// TIA Portal V15.1 export
// export: Created 2024-06-21T08:41:19.1954303Z, ExportSetting WithDefaults, DisplayName Totally Integrated Automation Portal, DisplayVersion V15.1 Update 5, DisplayName TIA Portal Openness, DisplayVersion V15.1 Update 5, DisplayName SINAMICS Startdrive Advanced, DisplayVersion V15.1, DisplayName G130, G150, S120, S150, SINAMICS MV, S210, DisplayVersion V15.1, DisplayName G110M, G120, G120C, G120D, G120P, DisplayVersion V15.1, DisplayName STEP 7 Professional, DisplayVersion V15.1 Update 5, DisplayName STEP 7 Safety, DisplayVersion V15.1, DisplayName WinCC Professional, DisplayVersion V15.1 Update 5, DisplayName SIMATIC Visualization Architect, DisplayVersion V15.1
FUNCTION_BLOCK "LGBHoist5Pos-MoviProPN"   // FB6695, FBD
TITLE = LGBMovUnit4Pos-MoviProPN / LGBHoist5Pos-MoviProPN
{ S7_Optimized_Access := 'TRUE' }
AUTHOR : VCC
VERSION : 0.0.0.0
// ============================================================================
// This module is used in applications with a EPOS controlled by a SEW MoviPro frequency converter.
// ============================================================================
// stored: AutoNumber false, IsIECCheckEnabled false, IsRetainMemResEnabled false, MemoryReserve 100, SetENOAutomatically False, UDAEnableTagReadback false
   VAR_INPUT
      I_BeltCheckSensor1 { ExternalAccessible := 'False'; ExternalVisible := 'False'; ExternalWritable := 'False'} : Bool;   // Belt check sensor
      I_BeltCheckSensor2 { ExternalAccessible := 'False'; ExternalVisible := 'False'; ExternalWritable := 'False'} : Bool;   // Belt check sensor
      I_ClutchDetection1 { ExternalAccessible := 'False'; ExternalVisible := 'False'; ExternalWritable := 'False'} : Bool;   // Clutch detection
      I_ClutchDetection2 { ExternalAccessible := 'False'; ExternalVisible := 'False'; ExternalWritable := 'False'} : Bool;   // Clutch detection
      I_Position1Begin { ExternalAccessible := 'False'; ExternalVisible := 'False'; ExternalWritable := 'False'} : Bool;   // Start Move To Position
      I_Position2Begin { ExternalAccessible := 'False'; ExternalVisible := 'False'; ExternalWritable := 'False'} : Bool;   // Start Move To Position
      I_Position3Begin { ExternalAccessible := 'False'; ExternalVisible := 'False'; ExternalWritable := 'False'} : Bool;   // Start Move To Position
      I_Position4Begin { ExternalAccessible := 'False'; ExternalVisible := 'False'; ExternalWritable := 'False'} : Bool;   // Start Move To Position
      I_Position5Begin { ExternalAccessible := 'False'; ExternalVisible := 'False'; ExternalWritable := 'False'} : Bool;   // Start Move To Position
      I_PositionMaintenanceBegin { ExternalAccessible := 'False'; ExternalVisible := 'False'; ExternalWritable := 'False'} : Bool;   // Start Move To Position / Start Move To Position Maintenance
      I_InterlockPos1 { ExternalAccessible := 'False'; ExternalVisible := 'False'; ExternalWritable := 'False'} : Bool;   // Interlock Pos1
      I_InterlockPos2 { ExternalAccessible := 'False'; ExternalVisible := 'False'; ExternalWritable := 'False'} : Bool;   // Interlock Pos2
      I_InterlockPos3 { ExternalAccessible := 'False'; ExternalVisible := 'False'; ExternalWritable := 'False'} : Bool;   // Interlock Pos3
      I_InterlockPos4 { ExternalAccessible := 'False'; ExternalVisible := 'False'; ExternalWritable := 'False'} : Bool;   // Interlock Pos4
      I_InterlockPos5 { ExternalAccessible := 'False'; ExternalVisible := 'False'; ExternalWritable := 'False'} : Bool;   // Interlock Pos4 / Interlock Pos5
      I_InterlockPosMaintenance { ExternalAccessible := 'False'; ExternalVisible := 'False'; ExternalWritable := 'False'} : Bool;   // Interlock Pos4 / Interlock Pos Maintenance
      I_InterlockJog { ExternalAccessible := 'False'; ExternalVisible := 'False'; ExternalWritable := 'False'} : Bool;   // Interlock Jog -/+ / Interlock jog set
      I_InterlockReferencing { ExternalAccessible := 'False'; ExternalVisible := 'False'; ExternalWritable := 'False'} : Bool;   // Interlock Referencing / Interlock jog set
      I_LocalPBSet { ExternalAccessible := 'False'; ExternalVisible := 'False'; ExternalWritable := 'False'} : Bool;   // Push button for manual movememt (on local panel)
      I_LocalPBRes { ExternalAccessible := 'False'; ExternalVisible := 'False'; ExternalWritable := 'False'} : Bool;   // Push button for manual movememt Reset(on local panel)
      I_MotorProtection { ExternalAccessible := 'False'; ExternalVisible := 'False'; ExternalWritable := 'False'} : Bool;   // Motor protection
      I_ReleaseBrake { ExternalAccessible := 'False'; ExternalVisible := 'False'; ExternalWritable := 'False'} : Bool;   // Release brake
      I_Distance { ExternalAccessible := 'False'; ExternalVisible := 'False'; ExternalWritable := 'False'} : DInt;   // Current distance / Current distance in the current resolution under consideration of offset. Depending on resolution, one digit corresponds to 0.1 to 100 mm.
      I_SafetyOk { ExternalAccessible := 'False'; ExternalVisible := 'False'; ExternalWritable := 'False'} : Bool;   // Safety Ok
      I_MotionStopOk { ExternalAccessible := 'False'; ExternalVisible := 'False'; ExternalWritable := 'False'} : Bool;   // Safety Ok / The motion stop is Ok
      I_AutoSpeed { ExternalAccessible := 'False'; ExternalVisible := 'False'; ExternalWritable := 'False'} : Int;   // Auto speed Value
      I_ManualSpeed { ExternalAccessible := 'False'; ExternalVisible := 'False'; ExternalWritable := 'False'} : Int;   // Manual speed Value
      I_SafetyStatus { ExternalAccessible := 'False'; ExternalVisible := 'False'; ExternalWritable := 'False'} : Word;   // Safety Status
      I_SafetyControl { ExternalAccessible := 'False'; ExternalVisible := 'False'; ExternalWritable := 'False'} : Word;   // Safety Control Word
   END_VAR
   VAR_OUTPUT
      O_Active { ExternalAccessible := 'False'; ExternalVisible := 'False'; ExternalWritable := 'False'} : Bool;   // Machine is active
      O_Position1Finished { ExternalAccessible := 'False'; ExternalVisible := 'False'; ExternalWritable := 'False'} : Bool;   // Position 1 finished
      O_Position2Finished { ExternalAccessible := 'False'; ExternalVisible := 'False'; ExternalWritable := 'False'} : Bool;   // Position 2 finished
      O_Position3Finished { ExternalAccessible := 'False'; ExternalVisible := 'False'; ExternalWritable := 'False'} : Bool;   // Position 3 finished
      O_Position4Finished { ExternalAccessible := 'False'; ExternalVisible := 'False'; ExternalWritable := 'False'} : Bool;   // Position 4 finished
      O_Position5Finished { ExternalAccessible := 'False'; ExternalVisible := 'False'; ExternalWritable := 'False'} : Bool;   // Position 4 finished / Position 5 finished
      O_PositionMaintenanceFinished { ExternalAccessible := 'False'; ExternalVisible := 'False'; ExternalWritable := 'False'} : Bool;   // Position 4 finished / Position Maintenance finished
      O_InPosition1 { ExternalAccessible := 'False'; ExternalVisible := 'False'; ExternalWritable := 'False'} : Bool;   // In Position 1
      O_InPosition2 { ExternalAccessible := 'False'; ExternalVisible := 'False'; ExternalWritable := 'False'} : Bool;   // In Position 2
      O_InPosition3 { ExternalAccessible := 'False'; ExternalVisible := 'False'; ExternalWritable := 'False'} : Bool;   // In Position 3
      O_InPosition4 { ExternalAccessible := 'False'; ExternalVisible := 'False'; ExternalWritable := 'False'} : Bool;   // In Position 4
      O_InPosition5 { ExternalAccessible := 'False'; ExternalVisible := 'False'; ExternalWritable := 'False'} : Bool;   // In Position 4 / In Position 5
      O_InPositionMaintenance { ExternalAccessible := 'False'; ExternalVisible := 'False'; ExternalWritable := 'False'} : Bool;   // In Position 4 / In Position Maintenance
      O_ActualPosition { ExternalAccessible := 'False'; ExternalVisible := 'False'; ExternalWritable := 'False'} : DInt;   // Actual position
      O_LEDPosition1 { ExternalAccessible := 'False'; ExternalVisible := 'False'; ExternalWritable := 'False'} : Bool;   // Ledindication / Led indication for Position1
      O_LEDPosition2 { ExternalAccessible := 'False'; ExternalVisible := 'False'; ExternalWritable := 'False'} : Bool;   // Ledindication / Led indication for Position2
      O_LEDPosition3 { ExternalAccessible := 'False'; ExternalVisible := 'False'; ExternalWritable := 'False'} : Bool;   // Ledindication / Led indication for Position3
      O_LEDPosition4 { ExternalAccessible := 'False'; ExternalVisible := 'False'; ExternalWritable := 'False'} : Bool;   // Ledindication / Led indication for Position4
      O_LEDPosition5 { ExternalAccessible := 'False'; ExternalVisible := 'False'; ExternalWritable := 'False'} : Bool;   // Ledindication / Led indication for Position5
      O_AlarmABCondition { ExternalAccessible := 'False'; ExternalVisible := 'False'; ExternalWritable := 'False'} : Bool;   // Alarm AB condition
      O_AlarmA { ExternalAccessible := 'False'; ExternalVisible := 'False'; ExternalWritable := 'False'} : Bool;   // Summation Alarm A
      O_AlarmB { ExternalAccessible := 'False'; ExternalVisible := 'False'; ExternalWritable := 'False'} : Bool;   // Summation Alarm B
      O_AlarmC { ExternalAccessible := 'False'; ExternalVisible := 'False'; ExternalWritable := 'False'} : Bool;   // Summation Alarm C
      O_AlarmD { ExternalAccessible := 'False'; ExternalVisible := 'False'; ExternalWritable := 'False'} : Bool;   // Summation Alarm D
      H_AlarmDWord { ExternalAccessible := 'False'; ExternalVisible := 'False'; ExternalWritable := 'False'} : DWord;   // HMI Animation of the alarms
      H_AlarmDWord2 { ExternalAccessible := 'False'; ExternalVisible := 'False'; ExternalWritable := 'False'} : DWord;   // HMI Animation of the alarms
   END_VAR
   VAR_IN_OUT
      IO_Modes : "Modes";   // Modes
      H_HMI : "H_HMI";   // Animation
      "H_GBHoist5Pos-MoviProPN" : "H_GBHoist5Pos-MoviProPN";   // Animation
      C_Config : "Hoist5Pos-MoviProPNConfig";   // Config
   END_VAR
   VAR
      AA_MotorProtection { ExternalAccessible := 'False'; ExternalVisible := 'False'; ExternalWritable := 'False'} : Bool;   // Motorprotection Tripped / Motorprotection Not Ok
      AA_SafetySwitch { ExternalAccessible := 'False'; ExternalVisible := 'False'; ExternalWritable := 'False'} : Bool;   // Safety Switch Not Ok
      AB_STO { ExternalAccessible := 'False'; ExternalVisible := 'False'; ExternalWritable := 'False'} : Bool;   // Safety Switch Not Ok / Safety output to drive is active but no response from drive that the safety is ok
      AB_DriveNoResponse { ExternalAccessible := 'False'; ExternalVisible := 'False'; ExternalWritable := 'False'} : Bool;   // Alarm Frequency Control / Alarm Frequency Control - No Responce from Drive (live bit)
      AB_DriveAlarm { ExternalAccessible := 'False'; ExternalVisible := 'False'; ExternalWritable := 'False'} : Bool;   // Frequency Control / Alarm Frequency Control
      AD_DriveWarning { ExternalAccessible := 'False'; ExternalVisible := 'False'; ExternalWritable := 'False'} : Bool;   // Warning Frequency Control / Warning
      AA_BeltCheck1 { ExternalAccessible := 'False'; ExternalVisible := 'False'; ExternalWritable := 'False'} : Bool;   // Remkontroll 1 / Belt Control Detection 1
      AA_BeltCheck2 { ExternalAccessible := 'False'; ExternalVisible := 'False'; ExternalWritable := 'False'} : Bool;   // Remkontroll 2 / Belt Control Detection 2
      AB_ClutchDetection { ExternalAccessible := 'False'; ExternalVisible := 'False'; ExternalWritable := 'False'} : Bool;   // Remkontroll 2 / No or both clutches engaged
      AB_OverTravelSet { ExternalAccessible := 'False'; ExternalVisible := 'False'; ExternalWritable := 'False'} : Bool;   // Overtravel Set
      AB_OverTravelRes { ExternalAccessible := 'False'; ExternalVisible := 'False'; ExternalWritable := 'False'} : Bool;   // Overtravel Reset
      AB_EncDifference { ExternalAccessible := 'False'; ExternalVisible := 'False'; ExternalWritable := 'False'} : Bool;   // Profinet <-> SSI encoder difference alarm
      AC_OvtPos1 { ExternalAccessible := 'False'; ExternalVisible := 'False'; ExternalWritable := 'False'} : Bool;   // Timeout Pos 1 / TimeOut to Position 1
      AC_OvtPos2 { ExternalAccessible := 'False'; ExternalVisible := 'False'; ExternalWritable := 'False'} : Bool;   // Timeout Pos 2 / TimeOut to Position 2
      AC_OvtPos3 { ExternalAccessible := 'False'; ExternalVisible := 'False'; ExternalWritable := 'False'} : Bool;   // Timeout Pos 3 / TimeOut to Position 3
      AC_OvtPos4 { ExternalAccessible := 'False'; ExternalVisible := 'False'; ExternalWritable := 'False'} : Bool;   // Timeout Pos 4 / TimeOut to Position 4
      AC_OvtPos5 { ExternalAccessible := 'False'; ExternalVisible := 'False'; ExternalWritable := 'False'} : Bool;   // Timeout Pos 4 / TimeOut to Position 5
      AC_OvtPosMaintenance { ExternalAccessible := 'False'; ExternalVisible := 'False'; ExternalWritable := 'False'} : Bool;   // Timeout Pos 4 / TimeOut to Position Maintenance
      AC_KeepPos1 { ExternalAccessible := 'False'; ExternalVisible := 'False'; ExternalWritable := 'False'} : Bool;   // Position Supervision / Lost Position 1
      AC_KeepPos2 { ExternalAccessible := 'False'; ExternalVisible := 'False'; ExternalWritable := 'False'} : Bool;   // Position Supervision / Lost Position 2
      AC_KeepPos3 { ExternalAccessible := 'False'; ExternalVisible := 'False'; ExternalWritable := 'False'} : Bool;   // Position Supervision / Lost Position 3
      AC_KeepPos4 { ExternalAccessible := 'False'; ExternalVisible := 'False'; ExternalWritable := 'False'} : Bool;   // Position Supervision / Lost Position 4
      AC_KeepPos5 { ExternalAccessible := 'False'; ExternalVisible := 'False'; ExternalWritable := 'False'} : Bool;   // Position Supervision / Lost Position 5
      AD_IntlkPos1 { ExternalAccessible := 'False'; ExternalVisible := 'False'; ExternalWritable := 'False'} : Bool;   // Interlock Not Ok / Interlock Position 1
      AD_IntlkPos2 { ExternalAccessible := 'False'; ExternalVisible := 'False'; ExternalWritable := 'False'} : Bool;   // Interlock Not Ok / Interlock Position 2
      AD_IntlkPos3 { ExternalAccessible := 'False'; ExternalVisible := 'False'; ExternalWritable := 'False'} : Bool;   // Interlock Not Ok / Interlock Position 3
      AD_IntlkPos4 { ExternalAccessible := 'False'; ExternalVisible := 'False'; ExternalWritable := 'False'} : Bool;   // Interlock Not Ok / Interlock Position 4
      AD_IntlkPos5 { ExternalAccessible := 'False'; ExternalVisible := 'False'; ExternalWritable := 'False'} : Bool;   // Interlock Not Ok / Interlock Position 5
      AD_IntlkPosMaintenance { ExternalAccessible := 'False'; ExternalVisible := 'False'; ExternalWritable := 'False'} : Bool;   // Interlock Not Ok / Interlock Position Maintenance
      AD_IntrlJogMode { ExternalAccessible := 'False'; ExternalVisible := 'False'; ExternalWritable := 'False'} : Bool;   // Interlock Jog Mode / Interlock Not Ok for jog set
      AD_IntrlReferencing { ExternalAccessible := 'False'; ExternalVisible := 'False'; ExternalWritable := 'False'} : Bool;   // Interlock Referencing / Interlock Not Ok for jog set
      AD_JogModeActive { ExternalAccessible := 'False'; ExternalVisible := 'False'; ExternalWritable := 'False'} : Bool;   // Jog Mode is active
      AD_ReferencingActive { ExternalAccessible := 'False'; ExternalVisible := 'False'; ExternalWritable := 'False'} : Bool;   // Referencing is active
      AD_EmergencyModeActive { ExternalAccessible := 'False'; ExternalVisible := 'False'; ExternalWritable := 'False'} : Bool;   // Emergency Mode is active
      AD_MotionStop { ExternalAccessible := 'False'; ExternalVisible := 'False'; ExternalWritable := 'False'} : Bool;   // Motion Stop
      SafetyOk { ExternalAccessible := 'False'; ExternalVisible := 'False'; ExternalWritable := 'False'} : Bool;   // Safety Ok
      AlarmA { ExternalAccessible := 'False'; ExternalVisible := 'False'; ExternalWritable := 'False'} : Bool;   // Alarm A
      AlarmB { ExternalAccessible := 'False'; ExternalVisible := 'False'; ExternalWritable := 'False'} : Bool;   // Alarm B
      AlarmC { ExternalAccessible := 'False'; ExternalVisible := 'False'; ExternalWritable := 'False'} : Bool;   // Alarm C
      AlarmD { ExternalAccessible := 'False'; ExternalVisible := 'False'; ExternalWritable := 'False'} : Bool;   // Alarm D
      AlarmABCondition { ExternalAccessible := 'False'; ExternalVisible := 'False'; ExternalWritable := 'False'} : Bool;   // Alarm AB Condition
      Referencing { ExternalAccessible := 'False'; ExternalVisible := 'False'; ExternalWritable := 'False'} : Bool;   // Activate Calibration
      EmergencyMode { ExternalAccessible := 'False'; ExternalVisible := 'False'; ExternalWritable := 'False'} : Bool;   // Emergency mode (without encoder)
      DriveMode { ExternalAccessible := 'False'; ExternalVisible := 'False'; ExternalWritable := 'False'} : Bool;   // 1 = direct setpoint / 0 = Jogmode
      JogMode { ExternalAccessible := 'False'; ExternalVisible := 'False'; ExternalWritable := 'False'} : Bool;   // 1= jog mode / 0= normal mode
      EPosCmdPos1 { ExternalAccessible := 'False'; ExternalVisible := 'False'; ExternalWritable := 'False'} : Bool;   // Cmd Pos 1 Direction
      EPosCmdPos2 { ExternalAccessible := 'False'; ExternalVisible := 'False'; ExternalWritable := 'False'} : Bool;   // Cmd Pos 2 Direction
      EPosCmdPos3 { ExternalAccessible := 'False'; ExternalVisible := 'False'; ExternalWritable := 'False'} : Bool;   // Cmd Pos 3 Direction
      EPosCmdPos4 { ExternalAccessible := 'False'; ExternalVisible := 'False'; ExternalWritable := 'False'} : Bool;   // Cmd Pos 4 Direction
      EPosCmdPos5 { ExternalAccessible := 'False'; ExternalVisible := 'False'; ExternalWritable := 'False'} : Bool;   // Cmd Pos 5 Direction / Cmd Pos 4 Direction
      EPosCmdPosMaintenance { ExternalAccessible := 'False'; ExternalVisible := 'False'; ExternalWritable := 'False'} : Bool;   // Cmd Pos Maintenance Direction / Cmd Pos 4 Direction
      MotorLoopActive { ExternalAccessible := 'False'; ExternalVisible := 'False'; ExternalWritable := 'False'} : Bool;   // Motor Loop Active
      BeltCheck1AlmCond { ExternalAccessible := 'False'; ExternalVisible := 'False'; ExternalWritable := 'False'} : Bool;   // Belt check alarm condition
      BeltCheck2AlmCond { ExternalAccessible := 'False'; ExternalVisible := 'False'; ExternalWritable := 'False'} : Bool;   // Belt check alarm condition
      ClutchDetectionAlmCond { ExternalAccessible := 'False'; ExternalVisible := 'False'; ExternalWritable := 'False'} : Bool;   // Belt check alarm condition
      OverTravelSetAlmCond { ExternalAccessible := 'False'; ExternalVisible := 'False'; ExternalWritable := 'False'} : Bool;   // Overtravel set alarm condition
      OverTravelResAlmCond { ExternalAccessible := 'False'; ExternalVisible := 'False'; ExternalWritable := 'False'} : Bool;   // Overtravel reset alarm condition
      MotorLoopAlarmCond { ExternalAccessible := 'False'; ExternalVisible := 'False'; ExternalWritable := 'False'} : Bool;   // Motor loop alarm condition
      EncDifferenceAlmCond { ExternalAccessible := 'False'; ExternalVisible := 'False'; ExternalWritable := 'False'} : Bool;   // Belt check alarm condition / Encoder Diff alarm condition
      ManReqIndexPos1 { ExternalAccessible := 'False'; ExternalVisible := 'False'; ExternalWritable := 'False'} : Bool;   // Manual request position 1
      ManReqIndexPos2 { ExternalAccessible := 'False'; ExternalVisible := 'False'; ExternalWritable := 'False'} : Bool;   // Manual request position 2
      ManReqIndexPos3 { ExternalAccessible := 'False'; ExternalVisible := 'False'; ExternalWritable := 'False'} : Bool;   // Manual request position 3
      ManReqIndexPos4 { ExternalAccessible := 'False'; ExternalVisible := 'False'; ExternalWritable := 'False'} : Bool;   // Manual request position 4
      ManReqIndexPos5 { ExternalAccessible := 'False'; ExternalVisible := 'False'; ExternalWritable := 'False'} : Bool;   // Manual request position 5 / Manual request position 4
      ManReqIndexPosMaintenance { ExternalAccessible := 'False'; ExternalVisible := 'False'; ExternalWritable := 'False'} : Bool;   // Manual request position Maintenance / Manual request position 4
      CmdPos1 { ExternalAccessible := 'False'; ExternalVisible := 'False'; ExternalWritable := 'False'} : Bool;   // Index position 1 command
      CmdPos2 { ExternalAccessible := 'False'; ExternalVisible := 'False'; ExternalWritable := 'False'} : Bool;   // Index position 2 command
      CmdPos3 { ExternalAccessible := 'False'; ExternalVisible := 'False'; ExternalWritable := 'False'} : Bool;   // Index position 3 command
      CmdPos4 { ExternalAccessible := 'False'; ExternalVisible := 'False'; ExternalWritable := 'False'} : Bool;   // Index position 4 command
      CmdPos5 { ExternalAccessible := 'False'; ExternalVisible := 'False'; ExternalWritable := 'False'} : Bool;   // Index position 4 command / Index position 5 command
      CmdPosMaintenance { ExternalAccessible := 'False'; ExternalVisible := 'False'; ExternalWritable := 'False'} : Bool;   // Index position 4 command / Index position Maintenance command
   END_VAR
   VAR RETAIN
      InPos1 { ExternalAccessible := 'False'; ExternalVisible := 'False'; ExternalWritable := 'False'} : Bool;   // In position 1
      InPos2 { ExternalAccessible := 'False'; ExternalVisible := 'False'; ExternalWritable := 'False'} : Bool;   // In position 2
      InPos3 { ExternalAccessible := 'False'; ExternalVisible := 'False'; ExternalWritable := 'False'} : Bool;   // In position 3
      InPos4 { ExternalAccessible := 'False'; ExternalVisible := 'False'; ExternalWritable := 'False'} : Bool;   // In position 4
      InPos5 { ExternalAccessible := 'False'; ExternalVisible := 'False'; ExternalWritable := 'False'} : Bool;   // In position 4 / In position 5
      InPosMaintenance { ExternalAccessible := 'False'; ExternalVisible := 'False'; ExternalWritable := 'False'} : Bool;   // In position 4 / In position Maintenance
   END_VAR
   VAR
      InterlockPos1 { ExternalAccessible := 'False'; ExternalVisible := 'False'; ExternalWritable := 'False'} : Bool;   // Interlock Pos1
      InterlockPos2 { ExternalAccessible := 'False'; ExternalVisible := 'False'; ExternalWritable := 'False'} : Bool;   // Interlock Pos2
      InterlockPos3 { ExternalAccessible := 'False'; ExternalVisible := 'False'; ExternalWritable := 'False'} : Bool;   // Interlock Pos3
      InterlockPos4 { ExternalAccessible := 'False'; ExternalVisible := 'False'; ExternalWritable := 'False'} : Bool;   // Interlock Pos4
      InterlockPos5 { ExternalAccessible := 'False'; ExternalVisible := 'False'; ExternalWritable := 'False'} : Bool;   // Interlock Pos4 / Interlock Pos5
      InterlockPosMaintenance { ExternalAccessible := 'False'; ExternalVisible := 'False'; ExternalWritable := 'False'} : Bool;   // Interlock Pos4 / Interlock PosMaintenance
      InterlockJog { ExternalAccessible := 'False'; ExternalVisible := 'False'; ExternalWritable := 'False'} : Bool;   // Interlock Jog -/+ / Interlock jog set
      InterlockReferencing { ExternalAccessible := 'False'; ExternalVisible := 'False'; ExternalWritable := 'False'} : Bool;   // Interlock Referencing / Interlock jog set
      ReadyForOperation { ExternalAccessible := 'False'; ExternalVisible := 'False'; ExternalWritable := 'False'} : Bool;   // Ready for operation
      EPOSInPosition { ExternalAccessible := 'False'; ExternalVisible := 'False'; ExternalWritable := 'False'} : Bool;   // Target Position reached
      AxisHomed { ExternalAccessible := 'False'; ExternalVisible := 'False'; ExternalWritable := 'False'} : Bool;   // Axis homed
      AxisMoving { ExternalAccessible := 'False'; ExternalVisible := 'False'; ExternalWritable := 'False'} : Bool;   // Axis moving in any direction
      InStandstill { ExternalAccessible := 'False'; ExternalVisible := 'False'; ExternalWritable := 'False'} : Bool;   // Axis in standstill
      Jog { ExternalAccessible := 'False'; ExternalVisible := 'False'; ExternalWritable := 'False'} : Bool;   // Activate Jog Mode
      Start { ExternalAccessible := 'False'; ExternalVisible := 'False'; ExternalWritable := 'False'} : Bool;   // Start command to motor
      SetpointSpeed { ExternalAccessible := 'False'; ExternalVisible := 'False'; ExternalWritable := 'False'} : Int;   // Setpoint speed
      LastCmd1 { ExternalAccessible := 'False'; ExternalVisible := 'False'; ExternalWritable := 'False'} : Bool;   // Last Command to Drive Is Pos 1
      LastCmd2 { ExternalAccessible := 'False'; ExternalVisible := 'False'; ExternalWritable := 'False'} : Bool;   // Last Command to Drive Is Pos 2
      LastCmd3 { ExternalAccessible := 'False'; ExternalVisible := 'False'; ExternalWritable := 'False'} : Bool;   // Last Command to Drive Is Pos 3
      LastCmd4 { ExternalAccessible := 'False'; ExternalVisible := 'False'; ExternalWritable := 'False'} : Bool;   // Last Command to Drive Is Pos 4
      LastCmd5 { ExternalAccessible := 'False'; ExternalVisible := 'False'; ExternalWritable := 'False'} : Bool;   // Last Command to Drive Is Pos 4 / Last Command to Drive Is Pos 5
      AlmCondKeepPos1 { ExternalAccessible := 'False'; ExternalVisible := 'False'; ExternalWritable := 'False'} : Bool;   // Alarm Condition Keep Position 1
      AlmCondKeepPos2 { ExternalAccessible := 'False'; ExternalVisible := 'False'; ExternalWritable := 'False'} : Bool;   // Alarm Condition Keep Position 2
      AlmCondKeepPos3 { ExternalAccessible := 'False'; ExternalVisible := 'False'; ExternalWritable := 'False'} : Bool;   // Alarm Condition Keep Position 3
      AlmCondKeepPos4 { ExternalAccessible := 'False'; ExternalVisible := 'False'; ExternalWritable := 'False'} : Bool;   // Alarm Condition Keep Position 4
      AlmCondKeepPos5 { ExternalAccessible := 'False'; ExternalVisible := 'False'; ExternalWritable := 'False'} : Bool;   // Alarm Condition Keep Position 4 / Alarm Condition Keep Position 5
      LowerLimit { ExternalAccessible := 'False'; ExternalVisible := 'False'; ExternalWritable := 'False'} : DInt;   // Lowest position
      UpperLimit { ExternalAccessible := 'False'; ExternalVisible := 'False'; ExternalWritable := 'False'} : DInt;   // Highest position
      SetpointPosition { ExternalAccessible := 'False'; ExternalVisible := 'False'; ExternalWritable := 'False'} : DInt;   // SetpointPosition
      OperatingMode { ExternalAccessible := 'False'; ExternalVisible := 'False'; ExternalWritable := 'False'} : USInt := 4;   // 0=Default, 1=Speed control, 2=Jog mode, 3=Referencing mode, 4=Positioning mode, 5=Positioning mode - touch probe, 6=Speed synchronization, 7=Emergency mode
      HWLSPositive { ExternalAccessible := 'False'; ExternalVisible := 'False'; ExternalWritable := 'False'} : Bool;   // Hardware limit switch from drive
      HWLSNegative { ExternalAccessible := 'False'; ExternalVisible := 'False'; ExternalWritable := 'False'} : Bool;   // Hardware limit switch from drive
      LockLocalPB { ExternalAccessible := 'False'; ExternalVisible := 'False'; ExternalWritable := 'False'} : Bool;   // Lock push button
      OvtMaxRunTime { ExternalAccessible := 'False'; ExternalVisible := 'False'; ExternalWritable := 'False'} : DInt;   // Alarm Value
      OvtMaxRunTimeCalc { ExternalAccessible := 'False'; ExternalVisible := 'False'; ExternalWritable := 'False'} : DInt;   // Alarm Value
      LastSetpointPosition { ExternalAccessible := 'False'; ExternalVisible := 'False'; ExternalWritable := 'False'} : DInt;
      DiffSetpointPosition { ExternalAccessible := 'False'; ExternalVisible := 'False'; ExternalWritable := 'False'} : DInt;
      H_Referencing { ExternalAccessible := 'False'; ExternalVisible := 'False'; ExternalWritable := 'False'} : Bool;   // Activate referencing / HMI Command - Activate referencing
      H_EmergencyMode { ExternalAccessible := 'False'; ExternalVisible := 'False'; ExternalWritable := 'False'} : Bool;   // Activate emergency mode / HMI Command - Activate emergency mode
      H_JogMode { ExternalAccessible := 'False'; ExternalVisible := 'False'; ExternalWritable := 'False'} : Bool;   // Activate Jog Mode / HMI Command - Activate Jog Mode
      H_CmdPos1 { ExternalAccessible := 'False'; ExternalVisible := 'False'; ExternalWritable := 'False'} : Bool;   // Temp / HMI Command - To Pos1
      H_CmdPos2 { ExternalAccessible := 'False'; ExternalVisible := 'False'; ExternalWritable := 'False'} : Bool;   // Temp / HMI Command - To Pos2
      H_CmdPos3 { ExternalAccessible := 'False'; ExternalVisible := 'False'; ExternalWritable := 'False'} : Bool;   // Temp / HMI Command - To Pos3
      H_CmdPos4 { ExternalAccessible := 'False'; ExternalVisible := 'False'; ExternalWritable := 'False'} : Bool;   // Temp / HMI Command - To Pos4
      H_CmdPos5 { ExternalAccessible := 'False'; ExternalVisible := 'False'; ExternalWritable := 'False'} : Bool;   // Temp / HMI Command - To Pos5
      H_CmdPosMaintenance { ExternalAccessible := 'False'; ExternalVisible := 'False'; ExternalWritable := 'False'} : Bool;   // Temp / HMI Command - To Maintenance Pos
      _Motor { ExternalAccessible := 'False'; ExternalVisible := 'False'; ExternalWritable := 'False'} : "LGBMotorEPos-MoviProPN";   // FB
      _OvertimePos1 { ExternalAccessible := 'False'; ExternalVisible := 'False'; ExternalWritable := 'False'} : "LTimer";   // FB
      _OvertimePos2 { ExternalAccessible := 'False'; ExternalVisible := 'False'; ExternalWritable := 'False'} : "LTimer";   // FB
      _OvertimePos3 { ExternalAccessible := 'False'; ExternalVisible := 'False'; ExternalWritable := 'False'} : "LTimer";   // FB
      _OvertimePos4 { ExternalAccessible := 'False'; ExternalVisible := 'False'; ExternalWritable := 'False'} : "LTimer";   // FB
      _OvertimePos5 { ExternalAccessible := 'False'; ExternalVisible := 'False'; ExternalWritable := 'False'} : "LTimer";   // FB
      _OvertimePosMaintenance { ExternalAccessible := 'False'; ExternalVisible := 'False'; ExternalWritable := 'False'} : "LTimer";   // FB
      _BeltCheck1 { ExternalAccessible := 'False'; ExternalVisible := 'False'; ExternalWritable := 'False'} : "L1AlarmMultiIn";   // FB
      _BeltCheck2 { ExternalAccessible := 'False'; ExternalVisible := 'False'; ExternalWritable := 'False'} : "L1AlarmMultiIn";   // FB
      _ClutchDetecion { ExternalAccessible := 'False'; ExternalVisible := 'False'; ExternalWritable := 'False'} : "L1AlarmMultiIn";   // FB
      _OverTravelSet { ExternalAccessible := 'False'; ExternalVisible := 'False'; ExternalWritable := 'False'} : "L1AlarmMultiIn";   // FB
      _OverTravelRes { ExternalAccessible := 'False'; ExternalVisible := 'False'; ExternalWritable := 'False'} : "L1AlarmMultiIn";   // FB
      _KeepPositionPos1 { ExternalAccessible := 'False'; ExternalVisible := 'False'; ExternalWritable := 'False'} : "L1AlarmMultiIn";   // Keep Position Alarm Position 1 / FB
      _KeepPositionPos2 { ExternalAccessible := 'False'; ExternalVisible := 'False'; ExternalWritable := 'False'} : "L1AlarmMultiIn";   // Keep Position Alarm Position 2 / FB
      _KeepPositionPos3 { ExternalAccessible := 'False'; ExternalVisible := 'False'; ExternalWritable := 'False'} : "L1AlarmMultiIn";   // Keep Position Alarm Position 3 / FB
      _KeepPositionPos4 { ExternalAccessible := 'False'; ExternalVisible := 'False'; ExternalWritable := 'False'} : "L1AlarmMultiIn";   // Keep Position Alarm Position 4 / FB
      _KeepPositionPos5 { ExternalAccessible := 'False'; ExternalVisible := 'False'; ExternalWritable := 'False'} : "L1AlarmMultiIn";   // Keep Position Alarm Position 4 / FB
      _EncDifference { ExternalAccessible := 'False'; ExternalVisible := 'False'; ExternalWritable := 'False'} : "L1AlarmMultiIn";   // FB
      Edge { ExternalAccessible := 'False'; ExternalVisible := 'False'; ExternalWritable := 'False'} : Array[0..20] of Bool;   // Flank
      T_DelayPB { ExternalAccessible := 'False'; ExternalVisible := 'False'; ExternalWritable := 'False'} : TON_TIME;   // Timer
      T_EncValueSTO { ExternalAccessible := 'False'; ExternalVisible := 'False'; ExternalWritable := 'False'} : TON_TIME;   // Timer
      T_EncValueError { ExternalAccessible := 'False'; ExternalVisible := 'False'; ExternalWritable := 'False'} : TON_TIME;   // Timer
   END_VAR
   VAR_TEMP
      NotUsedH_HMI : "H_HMI";   // Animation
      tTolerance : DInt;   // Tolerance for servo in Position
      tMinTolerancePos1 : DInt;   // Min tolerance for Position
      tMaxTolerancePos1 : DInt;   // Max tolerance for Position
      tMinTolerancePos2 : DInt;   // Min tolerance for Position
      tMaxTolerancePos2 : DInt;   // Max tolerance for Position
      tMinTolerancePos3 : DInt;   // Min tolerance for Position
      tMaxTolerancePos3 : DInt;   // Max tolerance for Position
      tMinTolerancePos4 : DInt;   // Min tolerance for Position
      tMaxTolerancePos4 : DInt;   // Max tolerance for Position
      tMinTolerancePos5 : DInt;   // Min tolerance for Position
      tMaxTolerancePos5 : DInt;   // Max tolerance for Position
      tMinTolerancePosMaintenance : DInt;   // Min tolerance for Position
      tMaxTolerancePosMaintenance : DInt;   // Max tolerance for Position
      JogSet : Bool;   // Temp
      JogRes : Bool;   // Temp
      tPositionSet : DInt;
      tPositionReset : DInt;
      tUpperLimit : DInt;
      tLowerLimit : DInt;
      tOvertimePos : DInt;
   END_VAR
   VAR_TEMP   // added for the SCL form of the ladder/FBD networks
      _w1 : Bool;
      _w2 : Bool;
      _w3 : Bool;
      _w4 : Bool;
      _w5 : Bool;
   END_VAR
BEGIN

REGION Network 1: **** 1 - Inputs **** HMI Commands
   // Extract The Commands From HMI
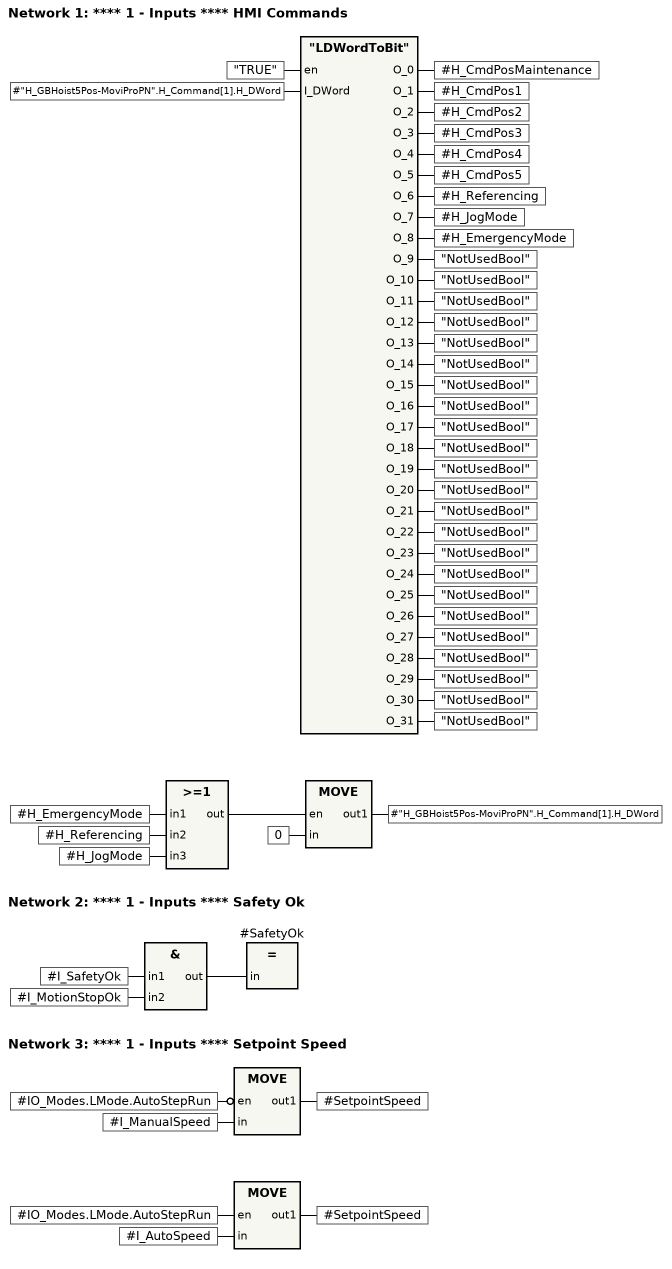
   IF "TRUE" THEN
       "LDWordToBit"(I_DWord := #"H_GBHoist5Pos-MoviProPN".H_Command[1].H_DWord,
                     O_0 => #H_CmdPosMaintenance,
                     O_1 => #H_CmdPos1,
                     O_2 => #H_CmdPos2,
                     O_3 => #H_CmdPos3,
                     O_4 => #H_CmdPos4,
                     O_5 => #H_CmdPos5,
                     O_6 => #H_Referencing,
                     O_7 => #H_JogMode,
                     O_8 => #H_EmergencyMode,
                     O_9 => "NotUsedBool",
                     O_10 => "NotUsedBool",
                     O_11 => "NotUsedBool",
                     O_12 => "NotUsedBool",
                     O_13 => "NotUsedBool",
                     O_14 => "NotUsedBool",
                     O_15 => "NotUsedBool",
                     O_16 => "NotUsedBool",
                     O_17 => "NotUsedBool",
                     O_18 => "NotUsedBool",
                     O_19 => "NotUsedBool",
                     O_20 => "NotUsedBool",
                     O_21 => "NotUsedBool",
                     O_22 => "NotUsedBool",
                     O_23 => "NotUsedBool",
                     O_24 => "NotUsedBool",
                     O_25 => "NotUsedBool",
                     O_26 => "NotUsedBool",
                     O_27 => "NotUsedBool",
                     O_28 => "NotUsedBool",
                     O_29 => "NotUsedBool",
                     O_30 => "NotUsedBool",
                     O_31 => "NotUsedBool");
   END_IF;
   IF #H_EmergencyMode OR #H_Referencing OR #H_JogMode THEN
       #"H_GBHoist5Pos-MoviProPN".H_Command[1].H_DWord := 0;
   END_IF;
END_REGION

REGION Network 2: **** 1 - Inputs **** Safety Ok
   #SafetyOk := #I_SafetyOk AND #I_MotionStopOk;
END_REGION

REGION Network 3: **** 1 - Inputs **** Setpoint Speed
   IF NOT #IO_Modes.LMode.AutoStepRun THEN #SetpointSpeed := #I_ManualSpeed; END_IF;
   IF #IO_Modes.LMode.AutoStepRun THEN #SetpointSpeed := #I_AutoSpeed; END_IF;
END_REGION

REGION Network 4: Calibrated Set / **** 1 - Input **** Ovt Values / **** 1 - Inputs **** Ovt Values / **** 1 - Input **** Overtime Values
   // Ovt Values
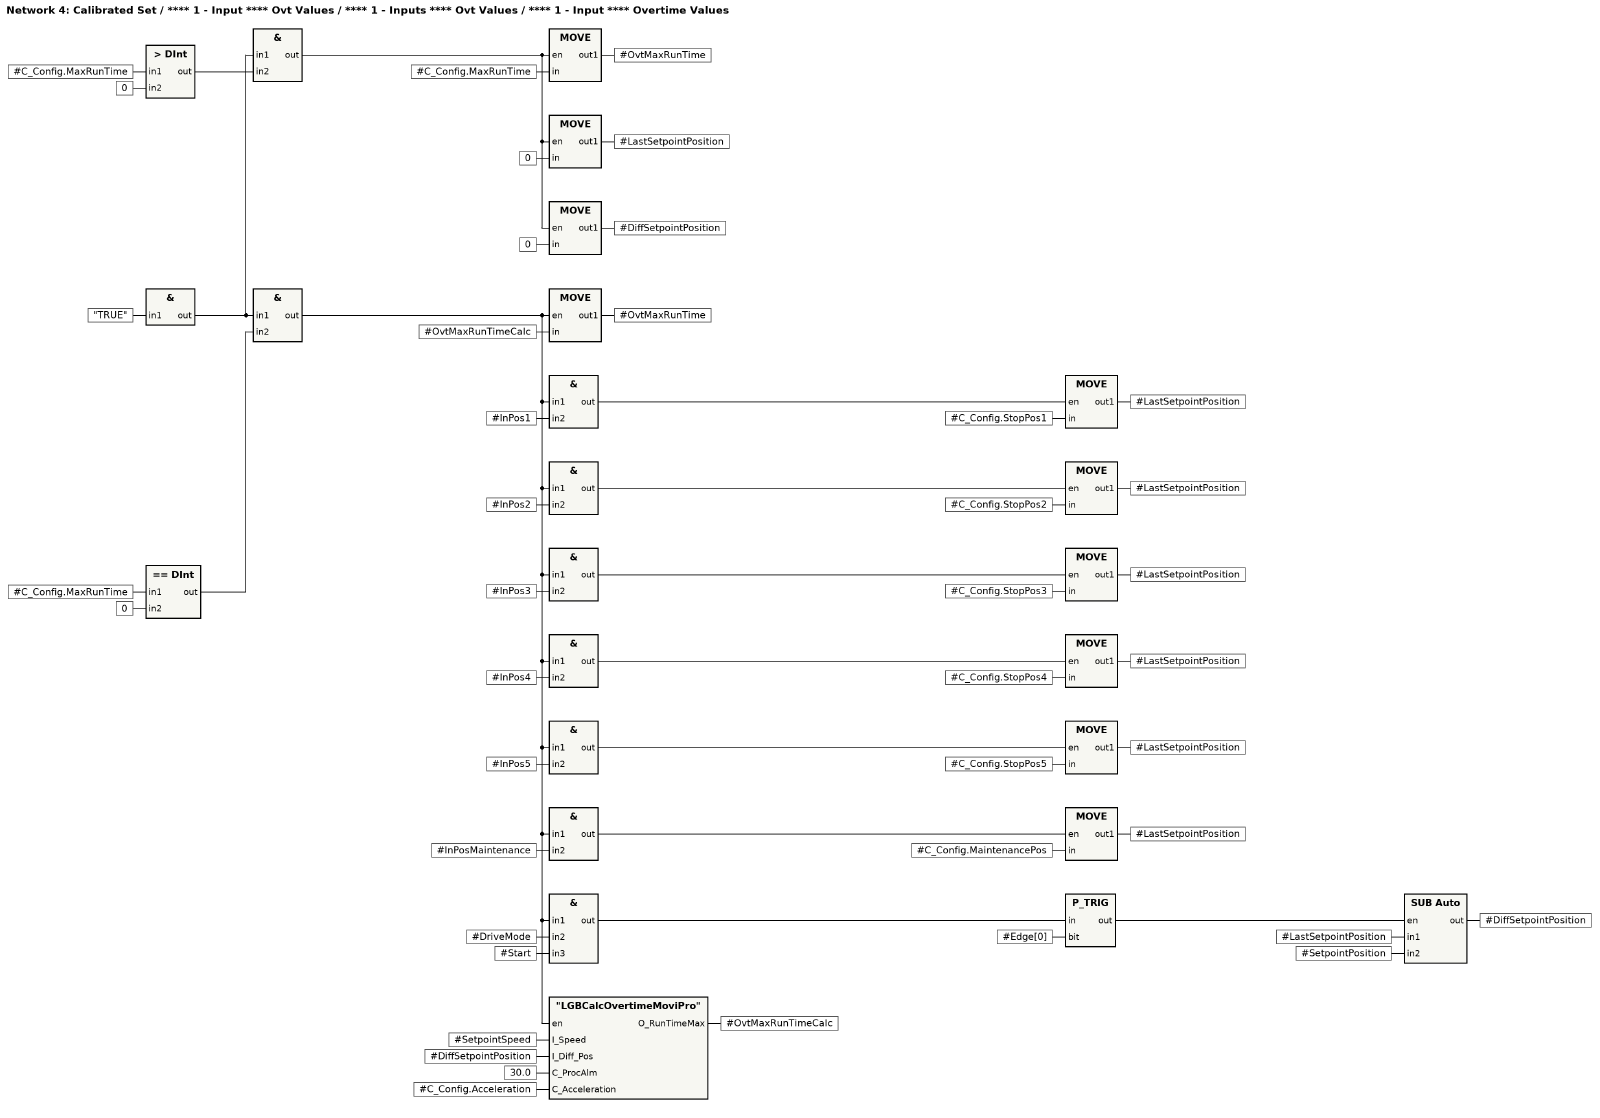
   IF "TRUE" AND (#C_Config.MaxRunTime > 0) THEN
       #OvtMaxRunTime := #C_Config.MaxRunTime;
       #LastSetpointPosition := 0;
       #DiffSetpointPosition := 0;
   END_IF;
   #_w1 := "TRUE" AND (#C_Config.MaxRunTime = 0);
   IF #_w1 THEN #OvtMaxRunTime := #OvtMaxRunTimeCalc; END_IF;
   IF #_w1 AND #InPos1 THEN #LastSetpointPosition := #C_Config.StopPos1; END_IF;
   IF #_w1 AND #InPos2 THEN #LastSetpointPosition := #C_Config.StopPos2; END_IF;
   IF #_w1 AND #InPos3 THEN #LastSetpointPosition := #C_Config.StopPos3; END_IF;
   IF #_w1 AND #InPos4 THEN #LastSetpointPosition := #C_Config.StopPos4; END_IF;
   IF #_w1 AND #InPos5 THEN #LastSetpointPosition := #C_Config.StopPos5; END_IF;
   IF #_w1 AND #InPosMaintenance THEN #LastSetpointPosition := #C_Config.MaintenancePos; END_IF;
   #_w2 := #_w1 AND #DriveMode AND #Start;
   #_w3 := #_w2 AND NOT #Edge[0];   // rising edge
   #Edge[0] := #_w2;
   IF #_w3 THEN #DiffSetpointPosition := #LastSetpointPosition - #SetpointPosition; END_IF;
   IF #_w1 THEN
       "LGBCalcOvertimeMoviPro"(I_Speed := #SetpointSpeed,
                               I_Diff_Pos := #DiffSetpointPosition,
                               C_ProcAlm := 30.0,
                               C_Acceleration := #C_Config.Acceleration,
                               O_RunTimeMax => #OvtMaxRunTimeCalc);
   END_IF;
END_REGION

REGION Network 5: **** 1 - Inputs **** Lock local PB on position
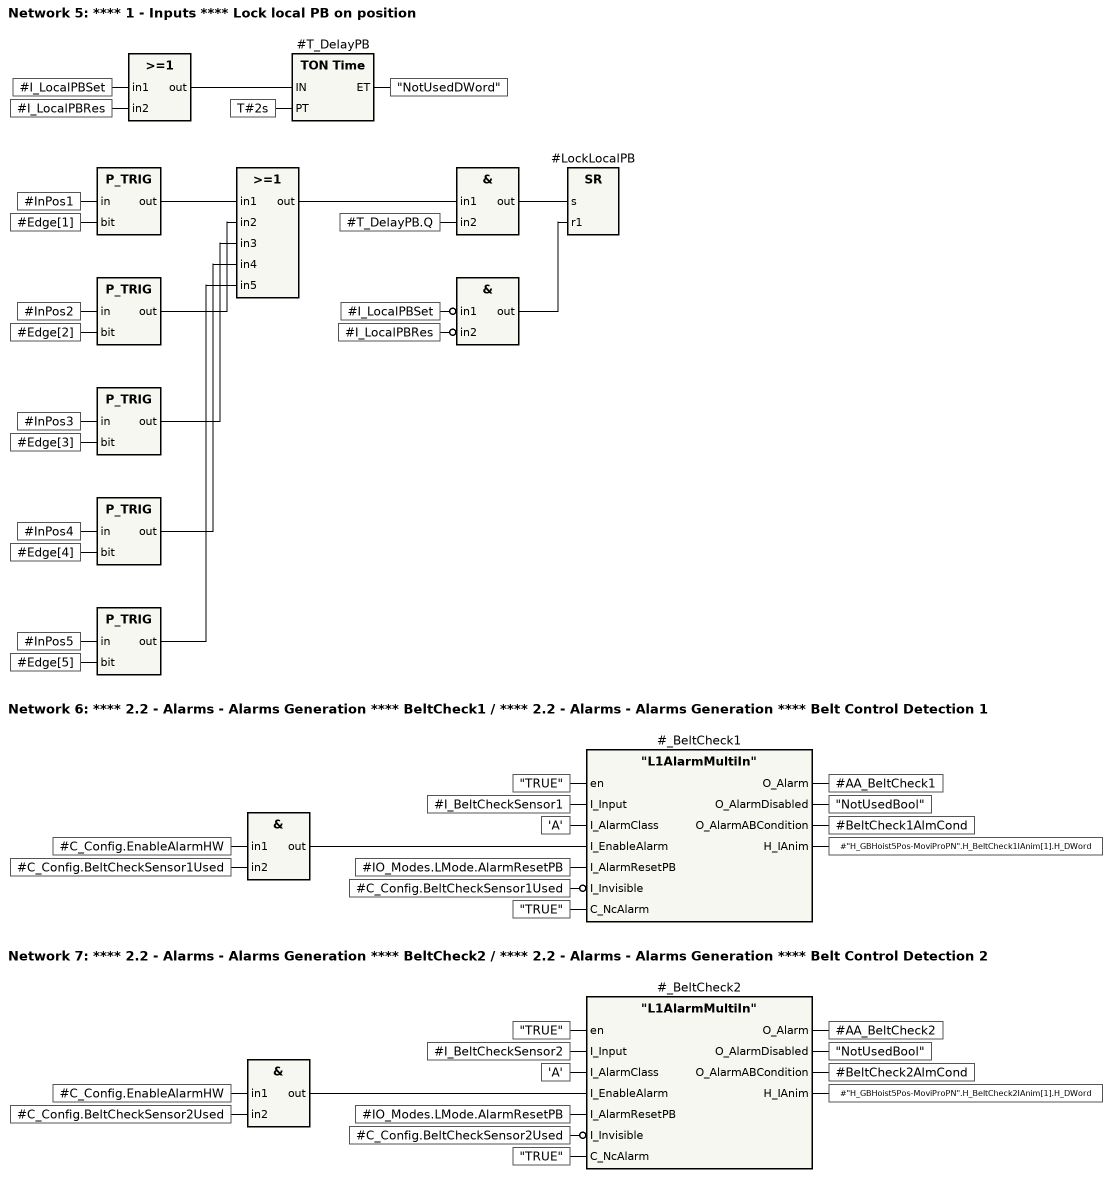
   #T_DelayPB(IN := #I_LocalPBSet OR #I_LocalPBRes, PT := T#2s, ET => "NotUsedDWord");   // TON
   #_w1 := #InPos1 AND NOT #Edge[1];   // rising edge
   #Edge[1] := #InPos1;
   #_w2 := #InPos2 AND NOT #Edge[2];   // rising edge
   #Edge[2] := #InPos2;
   #_w3 := #InPos3 AND NOT #Edge[3];   // rising edge
   #Edge[3] := #InPos3;
   #_w4 := #InPos4 AND NOT #Edge[4];   // rising edge
   #Edge[4] := #InPos4;
   #_w5 := #InPos5 AND NOT #Edge[5];   // rising edge
   #Edge[5] := #InPos5;
   IF (#_w1 OR #_w2 OR #_w3 OR #_w4 OR #_w5) AND #T_DelayPB.Q THEN
       #LockLocalPB := TRUE;   // SR flip-flop
   END_IF;
   IF NOT #I_LocalPBSet AND NOT #I_LocalPBRes THEN #LockLocalPB := FALSE; END_IF;
END_REGION

REGION Network 6: **** 2.2 - Alarms - Alarms Generation **** BeltCheck1 / **** 2.2 - Alarms - Alarms Generation **** Belt Control Detection 1
   // Alarm Belt check 1
   IF "TRUE" THEN
       #_BeltCheck1(I_Input := #I_BeltCheckSensor1,   // "L1AlarmMultiIn"
                    I_AlarmClass := 'A',
                    I_EnableAlarm := #C_Config.EnableAlarmHW AND #C_Config.BeltCheckSensor1Used,
                    I_AlarmResetPB := #IO_Modes.LMode.AlarmResetPB,
                    I_Invisible := NOT #C_Config.BeltCheckSensor1Used,
                    C_NcAlarm := "TRUE",
                    O_Alarm => #AA_BeltCheck1,
                    O_AlarmDisabled => "NotUsedBool",
                    O_AlarmABCondition => #BeltCheck1AlmCond,
                    H_IAnim => #"H_GBHoist5Pos-MoviProPN".H_BeltCheck1IAnim[1].H_DWord);
   END_IF;
END_REGION

REGION Network 7: **** 2.2 - Alarms - Alarms Generation **** BeltCheck2 / **** 2.2 - Alarms - Alarms Generation **** Belt Control Detection 2
   // Alarm Belt check 2
   IF "TRUE" THEN
       #_BeltCheck2(I_Input := #I_BeltCheckSensor2,   // "L1AlarmMultiIn"
                    I_AlarmClass := 'A',
                    I_EnableAlarm := #C_Config.EnableAlarmHW AND #C_Config.BeltCheckSensor2Used,
                    I_AlarmResetPB := #IO_Modes.LMode.AlarmResetPB,
                    I_Invisible := NOT #C_Config.BeltCheckSensor2Used,
                    C_NcAlarm := "TRUE",
                    O_Alarm => #AA_BeltCheck2,
                    O_AlarmDisabled => "NotUsedBool",
                    O_AlarmABCondition => #BeltCheck2AlmCond,
                    H_IAnim => #"H_GBHoist5Pos-MoviProPN".H_BeltCheck2IAnim[1].H_DWord);
   END_IF;
END_REGION

REGION Network 8: **** 2.2 - Alarms - Alarms Generation **** Clutch detections / **** 2.2 - Alarms - Alarms Generation **** No or both clutches engaged
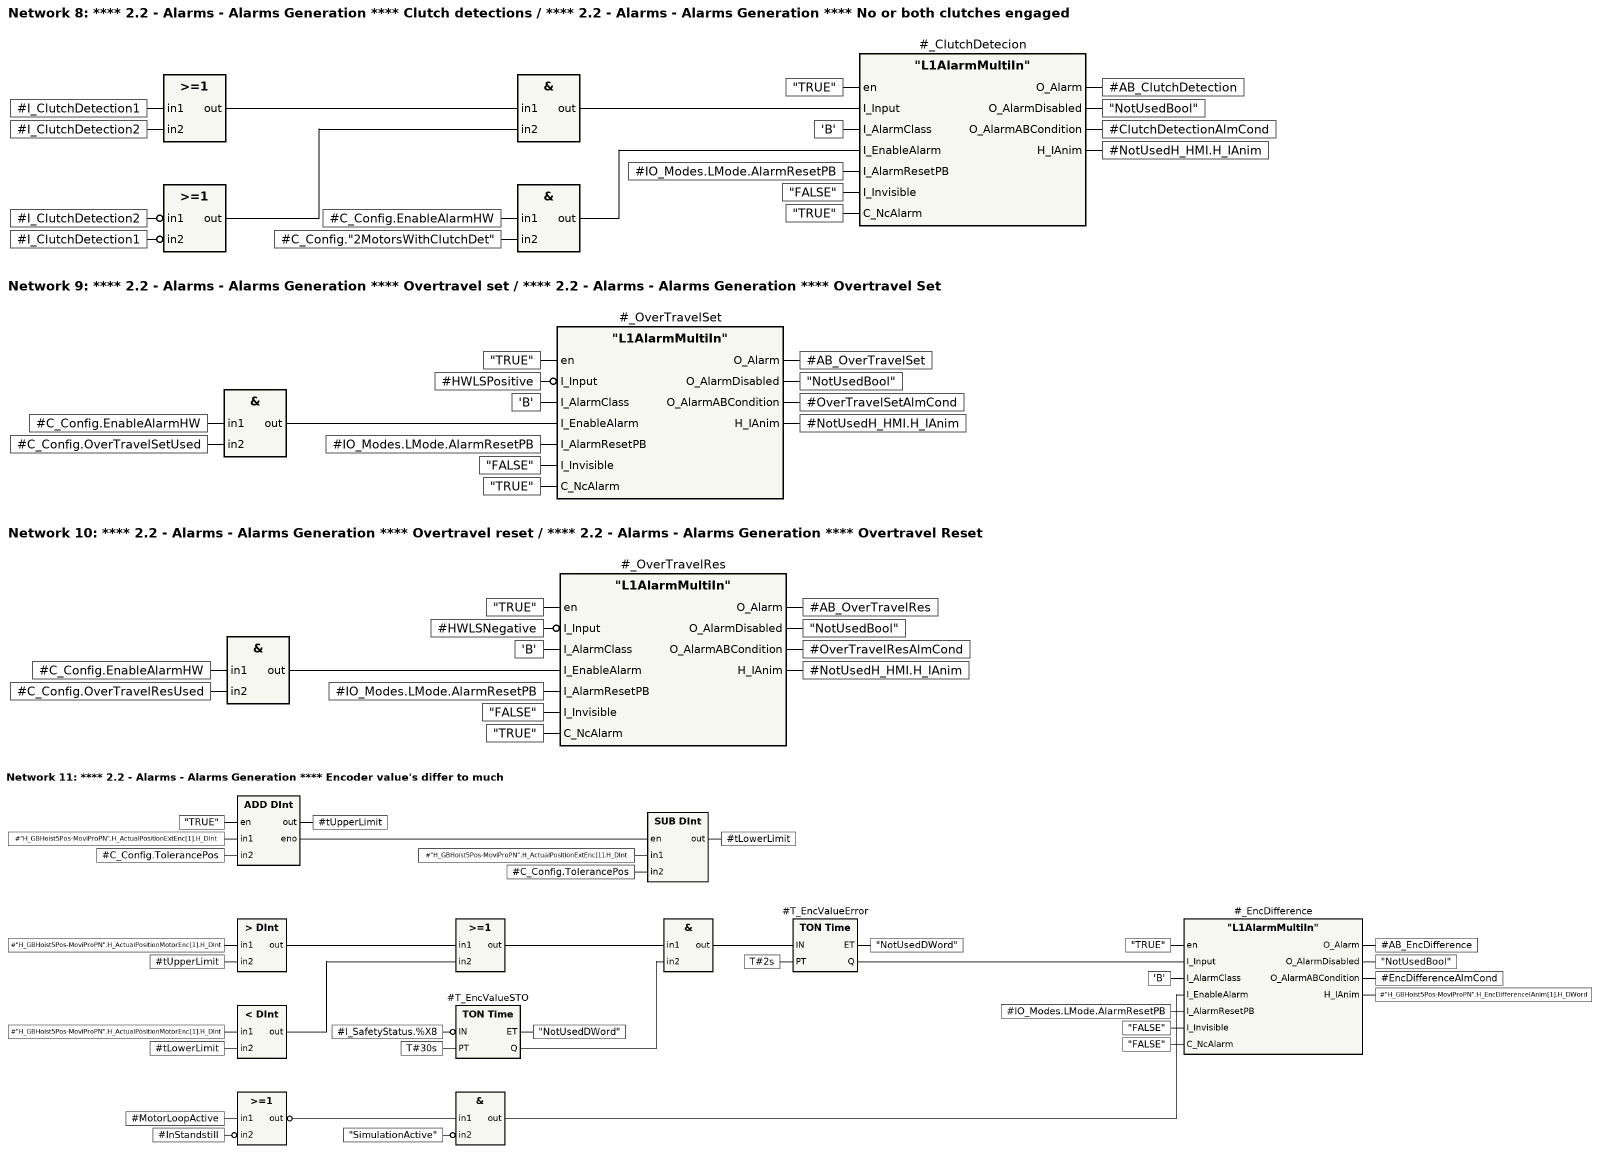
   IF "TRUE" THEN
       #_ClutchDetecion(I_Input := (#I_ClutchDetection1 OR #I_ClutchDetection2) AND (NOT #I_ClutchDetection2 OR NOT #I_ClutchDetection1),   // "L1AlarmMultiIn"
                        I_AlarmClass := 'B',
                        I_EnableAlarm := #C_Config.EnableAlarmHW AND #C_Config."2MotorsWithClutchDet",
                        I_AlarmResetPB := #IO_Modes.LMode.AlarmResetPB,
                        I_Invisible := "FALSE",
                        C_NcAlarm := "TRUE",
                        O_Alarm => #AB_ClutchDetection,
                        O_AlarmDisabled => "NotUsedBool",
                        O_AlarmABCondition => #ClutchDetectionAlmCond,
                        H_IAnim => #NotUsedH_HMI.H_IAnim);
   END_IF;
END_REGION

REGION Network 9: **** 2.2 - Alarms - Alarms Generation **** Overtravel set / **** 2.2 - Alarms - Alarms Generation **** Overtravel Set
   // Alarm Lift upper limit
   IF "TRUE" THEN
       #_OverTravelSet(I_Input := NOT #HWLSPositive,   // "L1AlarmMultiIn"
                       I_AlarmClass := 'B',
                       I_EnableAlarm := #C_Config.EnableAlarmHW AND #C_Config.OverTravelSetUsed,
                       I_AlarmResetPB := #IO_Modes.LMode.AlarmResetPB,
                       I_Invisible := "FALSE",
                       C_NcAlarm := "TRUE",
                       O_Alarm => #AB_OverTravelSet,
                       O_AlarmDisabled => "NotUsedBool",
                       O_AlarmABCondition => #OverTravelSetAlmCond,
                       H_IAnim => #NotUsedH_HMI.H_IAnim);
   END_IF;
END_REGION

REGION Network 10: **** 2.2 - Alarms - Alarms Generation **** Overtravel reset / **** 2.2 - Alarms - Alarms Generation **** Overtravel Reset
   // Alarm Lift upper limit
   IF "TRUE" THEN
       #_OverTravelRes(I_Input := NOT #HWLSNegative,   // "L1AlarmMultiIn"
                       I_AlarmClass := 'B',
                       I_EnableAlarm := #C_Config.EnableAlarmHW AND #C_Config.OverTravelResUsed,
                       I_AlarmResetPB := #IO_Modes.LMode.AlarmResetPB,
                       I_Invisible := "FALSE",
                       C_NcAlarm := "TRUE",
                       O_Alarm => #AB_OverTravelRes,
                       O_AlarmDisabled => "NotUsedBool",
                       O_AlarmABCondition => #OverTravelResAlmCond,
                       H_IAnim => #NotUsedH_HMI.H_IAnim);
   END_IF;
END_REGION

REGION Network 11: **** 2.2 - Alarms - Alarms Generation **** Encoder value's differ to much
   // Profinet <-> SSI encoder difference alarm
   IF "TRUE" THEN
       #tUpperLimit := #"H_GBHoist5Pos-MoviProPN".H_ActualPositionExtEnc[1].H_DInt + #C_Config.TolerancePos;
       #tLowerLimit := #"H_GBHoist5Pos-MoviProPN".H_ActualPositionExtEnc[1].H_DInt - #C_Config.TolerancePos;
   END_IF;
   #T_EncValueSTO(IN := NOT #I_SafetyStatus.%X8, PT := T#30s, ET => "NotUsedDWord");   // TON
   #T_EncValueError(IN := ((#"H_GBHoist5Pos-MoviProPN".H_ActualPositionMotorEnc[1].H_DInt > #tUpperLimit) OR (#"H_GBHoist5Pos-MoviProPN".H_ActualPositionMotorEnc[1].H_DInt < #tLowerLimit)) AND #T_EncValueSTO.Q,   // TON
                    PT := T#2s,
                    ET => "NotUsedDWord");
   IF "TRUE" THEN
       #_EncDifference(I_Input := #T_EncValueError.Q,   // "L1AlarmMultiIn"
                       I_AlarmClass := 'B',
                       I_EnableAlarm := NOT (#MotorLoopActive OR NOT #InStandstill) AND NOT "SimulationActive",
                       I_AlarmResetPB := #IO_Modes.LMode.AlarmResetPB,
                       I_Invisible := "FALSE",
                       C_NcAlarm := "FALSE",
                       O_Alarm => #AB_EncDifference,
                       O_AlarmDisabled => "NotUsedBool",
                       O_AlarmABCondition => #EncDifferenceAlmCond,
                       H_IAnim => #"H_GBHoist5Pos-MoviProPN".H_EncDifferenceIAnim[1].H_DWord);
   END_IF;
END_REGION

REGION Network 12: **** 2.2 - Alarms - Alarm Generation **** Delay-On timer Overtime Alarm Position 1 / **** 2.2 - Alarms - Alarm Generation **** TimeOut to Position 1
   // Delay-On timer Overtime Alarm Position 1
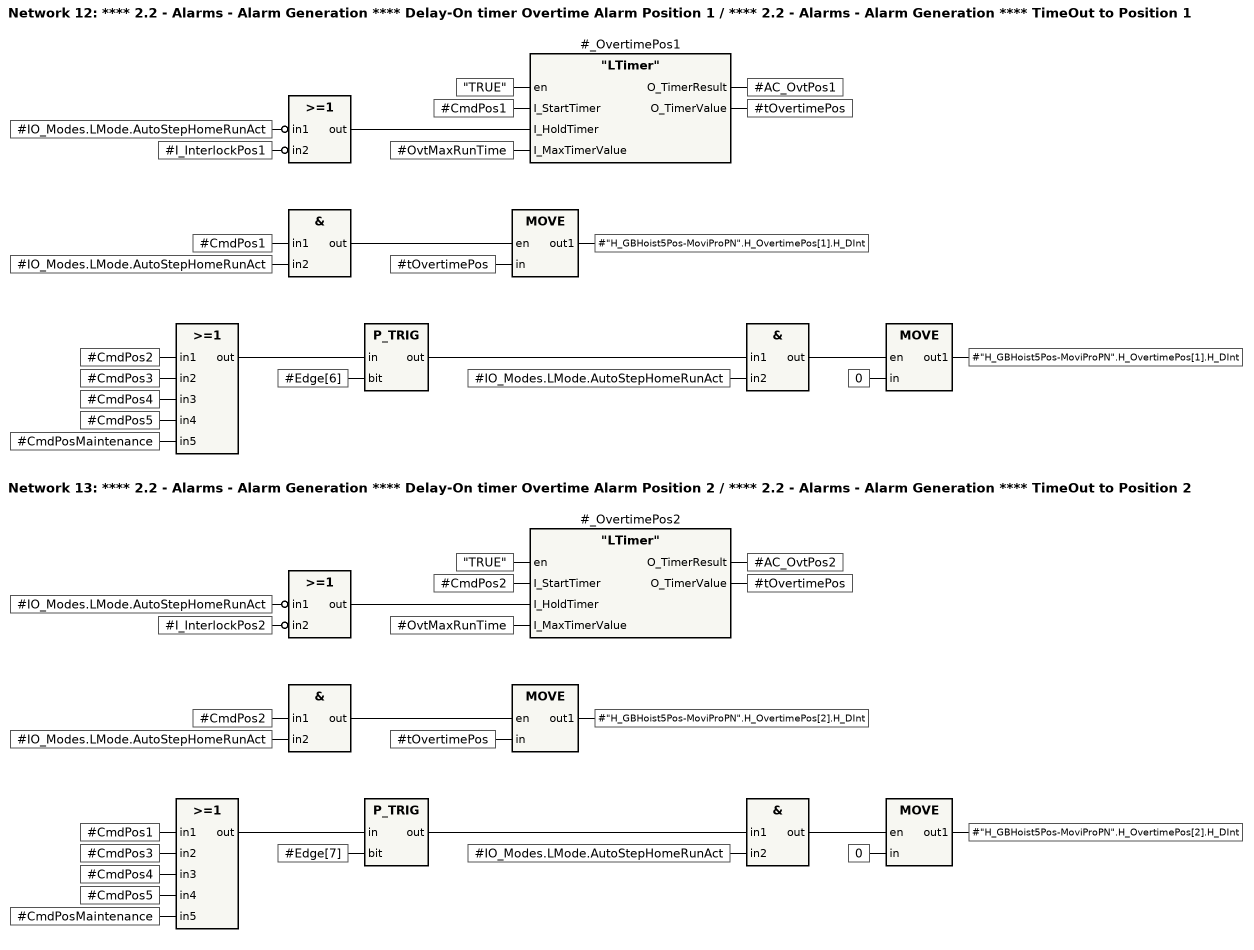
   IF "TRUE" THEN
       #_OvertimePos1(I_StartTimer := #CmdPos1,   // "LTimer"
                      I_HoldTimer := NOT #IO_Modes.LMode.AutoStepHomeRunAct OR NOT #I_InterlockPos1,
                      I_MaxTimerValue := #OvtMaxRunTime,
                      O_TimerResult => #AC_OvtPos1,
                      O_TimerValue => #tOvertimePos);
   END_IF;
   IF #CmdPos1 AND #IO_Modes.LMode.AutoStepHomeRunAct THEN
       #"H_GBHoist5Pos-MoviProPN".H_OvertimePos[1].H_DInt := #tOvertimePos;
   END_IF;
   #_w1 := #CmdPos2 OR #CmdPos3 OR #CmdPos4 OR #CmdPos5 OR #CmdPosMaintenance;
   #_w2 := #_w1 AND NOT #Edge[6];   // rising edge
   #Edge[6] := #_w1;
   IF #_w2 AND #IO_Modes.LMode.AutoStepHomeRunAct THEN
       #"H_GBHoist5Pos-MoviProPN".H_OvertimePos[1].H_DInt := 0;
   END_IF;
END_REGION

REGION Network 13: **** 2.2 - Alarms - Alarm Generation **** Delay-On timer Overtime Alarm Position 2 / **** 2.2 - Alarms - Alarm Generation **** TimeOut to Position 2
   // Delay-On timer Overtime Alarm Position 2
   IF "TRUE" THEN
       #_OvertimePos2(I_StartTimer := #CmdPos2,   // "LTimer"
                      I_HoldTimer := NOT #IO_Modes.LMode.AutoStepHomeRunAct OR NOT #I_InterlockPos2,
                      I_MaxTimerValue := #OvtMaxRunTime,
                      O_TimerResult => #AC_OvtPos2,
                      O_TimerValue => #tOvertimePos);
   END_IF;
   IF #CmdPos2 AND #IO_Modes.LMode.AutoStepHomeRunAct THEN
       #"H_GBHoist5Pos-MoviProPN".H_OvertimePos[2].H_DInt := #tOvertimePos;
   END_IF;
   #_w1 := #CmdPos1 OR #CmdPos3 OR #CmdPos4 OR #CmdPos5 OR #CmdPosMaintenance;
   #_w2 := #_w1 AND NOT #Edge[7];   // rising edge
   #Edge[7] := #_w1;
   IF #_w2 AND #IO_Modes.LMode.AutoStepHomeRunAct THEN
       #"H_GBHoist5Pos-MoviProPN".H_OvertimePos[2].H_DInt := 0;
   END_IF;
END_REGION

REGION Network 14: **** 2.2 - Alarms - Alarm Generation **** Delay-On timer Overtime Alarm Position 3 / **** 2.2 - Alarms - Alarm Generation **** TimeOut to Position 3
   // Delay-On timer Overtime Alarm Position 3
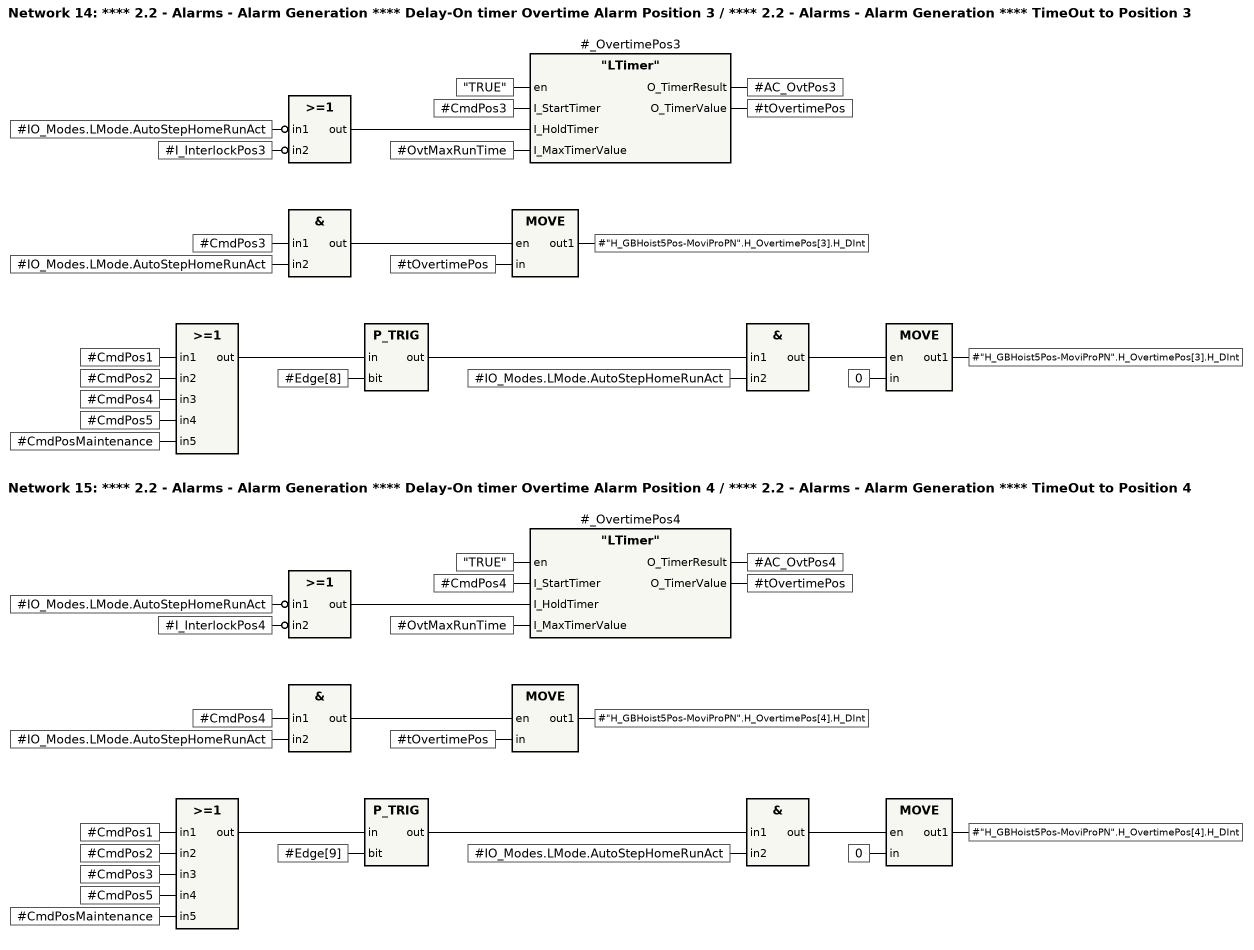
   IF "TRUE" THEN
       #_OvertimePos3(I_StartTimer := #CmdPos3,   // "LTimer"
                      I_HoldTimer := NOT #IO_Modes.LMode.AutoStepHomeRunAct OR NOT #I_InterlockPos3,
                      I_MaxTimerValue := #OvtMaxRunTime,
                      O_TimerResult => #AC_OvtPos3,
                      O_TimerValue => #tOvertimePos);
   END_IF;
   IF #CmdPos3 AND #IO_Modes.LMode.AutoStepHomeRunAct THEN
       #"H_GBHoist5Pos-MoviProPN".H_OvertimePos[3].H_DInt := #tOvertimePos;
   END_IF;
   #_w1 := #CmdPos1 OR #CmdPos2 OR #CmdPos4 OR #CmdPos5 OR #CmdPosMaintenance;
   #_w2 := #_w1 AND NOT #Edge[8];   // rising edge
   #Edge[8] := #_w1;
   IF #_w2 AND #IO_Modes.LMode.AutoStepHomeRunAct THEN
       #"H_GBHoist5Pos-MoviProPN".H_OvertimePos[3].H_DInt := 0;
   END_IF;
END_REGION

REGION Network 15: **** 2.2 - Alarms - Alarm Generation **** Delay-On timer Overtime Alarm Position 4 / **** 2.2 - Alarms - Alarm Generation **** TimeOut to Position 4
   // Delay-On timer Overtime Alarm Position 3
   IF "TRUE" THEN
       #_OvertimePos4(I_StartTimer := #CmdPos4,   // "LTimer"
                      I_HoldTimer := NOT #IO_Modes.LMode.AutoStepHomeRunAct OR NOT #I_InterlockPos4,
                      I_MaxTimerValue := #OvtMaxRunTime,
                      O_TimerResult => #AC_OvtPos4,
                      O_TimerValue => #tOvertimePos);
   END_IF;
   IF #CmdPos4 AND #IO_Modes.LMode.AutoStepHomeRunAct THEN
       #"H_GBHoist5Pos-MoviProPN".H_OvertimePos[4].H_DInt := #tOvertimePos;
   END_IF;
   #_w1 := #CmdPos1 OR #CmdPos2 OR #CmdPos3 OR #CmdPos5 OR #CmdPosMaintenance;
   #_w2 := #_w1 AND NOT #Edge[9];   // rising edge
   #Edge[9] := #_w1;
   IF #_w2 AND #IO_Modes.LMode.AutoStepHomeRunAct THEN
       #"H_GBHoist5Pos-MoviProPN".H_OvertimePos[4].H_DInt := 0;
   END_IF;
END_REGION

REGION Network 16: **** 2.2 - Alarms - Alarm Generation **** Delay-On timer Overtime Alarm Position 4 / **** 2.2 - Alarms - Alarm Generation **** TimeOut to Position 5
   // Delay-On timer Overtime Alarm Position 3
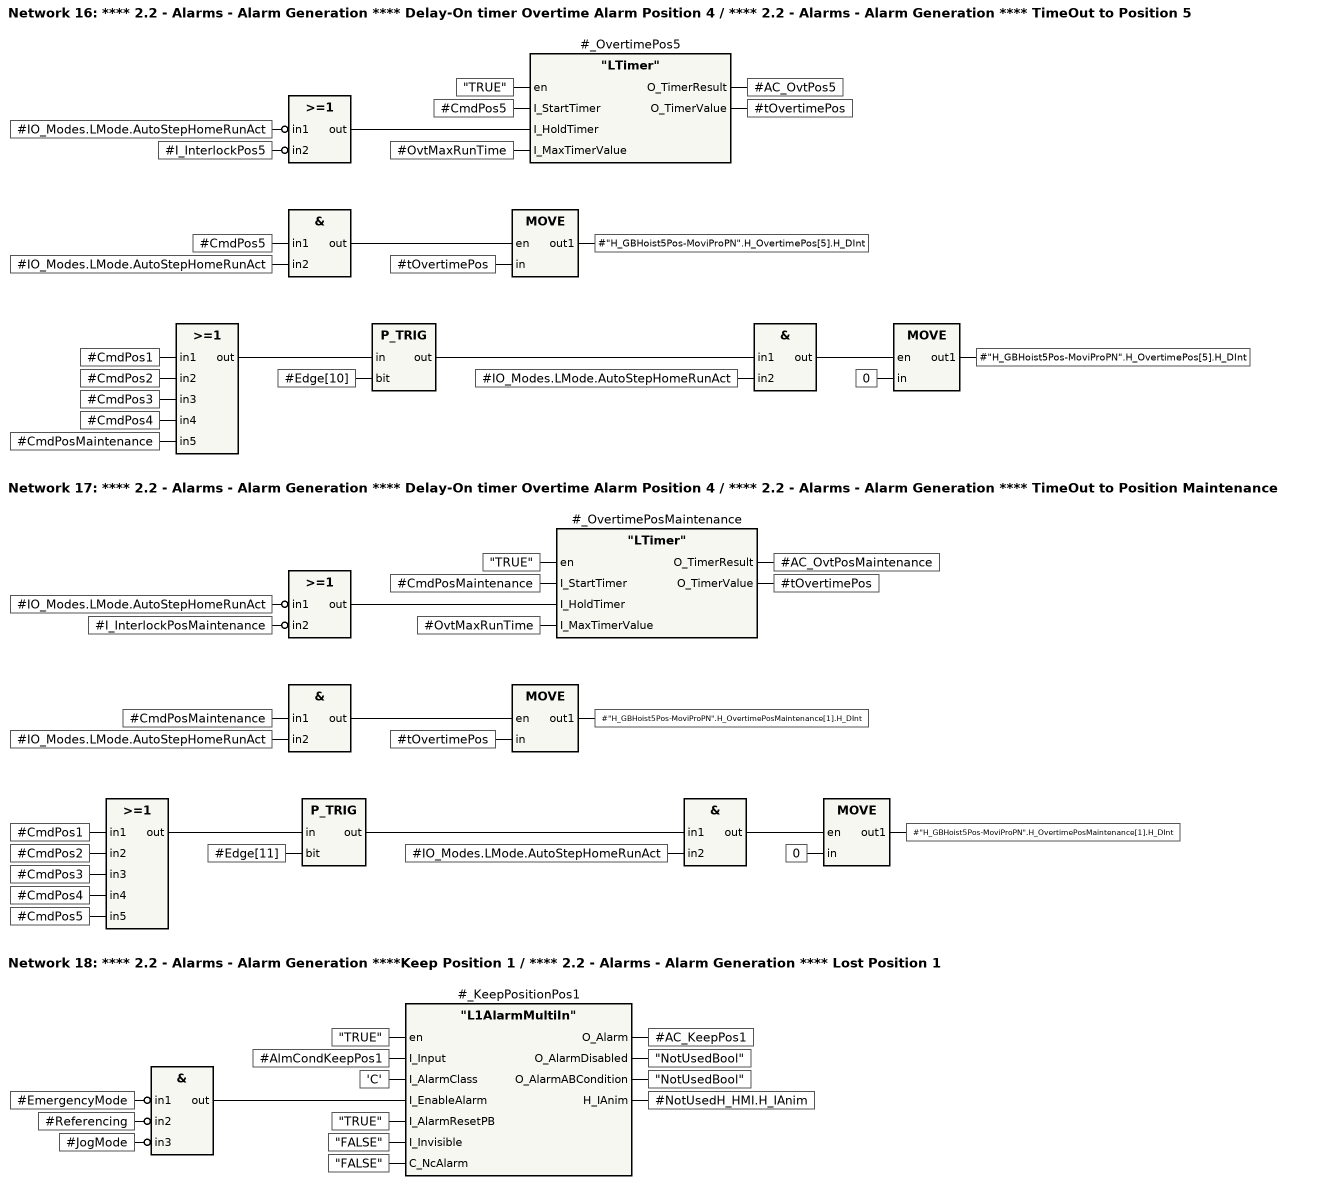
   IF "TRUE" THEN
       #_OvertimePos5(I_StartTimer := #CmdPos5,   // "LTimer"
                      I_HoldTimer := NOT #IO_Modes.LMode.AutoStepHomeRunAct OR NOT #I_InterlockPos5,
                      I_MaxTimerValue := #OvtMaxRunTime,
                      O_TimerResult => #AC_OvtPos5,
                      O_TimerValue => #tOvertimePos);
   END_IF;
   IF #CmdPos5 AND #IO_Modes.LMode.AutoStepHomeRunAct THEN
       #"H_GBHoist5Pos-MoviProPN".H_OvertimePos[5].H_DInt := #tOvertimePos;
   END_IF;
   #_w1 := #CmdPos1 OR #CmdPos2 OR #CmdPos3 OR #CmdPos4 OR #CmdPosMaintenance;
   #_w2 := #_w1 AND NOT #Edge[10];   // rising edge
   #Edge[10] := #_w1;
   IF #_w2 AND #IO_Modes.LMode.AutoStepHomeRunAct THEN
       #"H_GBHoist5Pos-MoviProPN".H_OvertimePos[5].H_DInt := 0;
   END_IF;
END_REGION

REGION Network 17: **** 2.2 - Alarms - Alarm Generation **** Delay-On timer Overtime Alarm Position 4 / **** 2.2 - Alarms - Alarm Generation **** TimeOut to Position Maintenance
   // Delay-On timer Overtime Alarm Position 3
   IF "TRUE" THEN
       #_OvertimePosMaintenance(I_StartTimer := #CmdPosMaintenance,   // "LTimer"
                               I_HoldTimer := NOT #IO_Modes.LMode.AutoStepHomeRunAct OR NOT #I_InterlockPosMaintenance,
                               I_MaxTimerValue := #OvtMaxRunTime,
                               O_TimerResult => #AC_OvtPosMaintenance,
                               O_TimerValue => #tOvertimePos);
   END_IF;
   IF #CmdPosMaintenance AND #IO_Modes.LMode.AutoStepHomeRunAct THEN
       #"H_GBHoist5Pos-MoviProPN".H_OvertimePosMaintenance[1].H_DInt := #tOvertimePos;
   END_IF;
   #_w1 := #CmdPos1 OR #CmdPos2 OR #CmdPos3 OR #CmdPos4 OR #CmdPos5;
   #_w2 := #_w1 AND NOT #Edge[11];   // rising edge
   #Edge[11] := #_w1;
   IF #_w2 AND #IO_Modes.LMode.AutoStepHomeRunAct THEN
       #"H_GBHoist5Pos-MoviProPN".H_OvertimePosMaintenance[1].H_DInt := 0;
   END_IF;
END_REGION

REGION Network 18: **** 2.2 - Alarms - Alarm Generation ****Keep Position 1 / **** 2.2 - Alarms - Alarm Generation **** Lost Position 1
   // Keep Position 1
   IF "TRUE" THEN
       #_KeepPositionPos1(I_Input := #AlmCondKeepPos1,   // "L1AlarmMultiIn"
                          I_AlarmClass := 'C',
                          I_EnableAlarm := NOT #EmergencyMode AND NOT #Referencing AND NOT #JogMode,
                          I_AlarmResetPB := "TRUE",
                          I_Invisible := "FALSE",
                          C_NcAlarm := "FALSE",
                          O_Alarm => #AC_KeepPos1,
                          O_AlarmDisabled => "NotUsedBool",
                          O_AlarmABCondition => "NotUsedBool",
                          H_IAnim => #NotUsedH_HMI.H_IAnim);
   END_IF;
END_REGION

REGION Network 19: **** 2.2 - Alarms - Alarm Generation ****Keep Position 2 / **** 2.2 - Alarms - Alarm Generation **** Lost Position 2
   // Keep Position 2
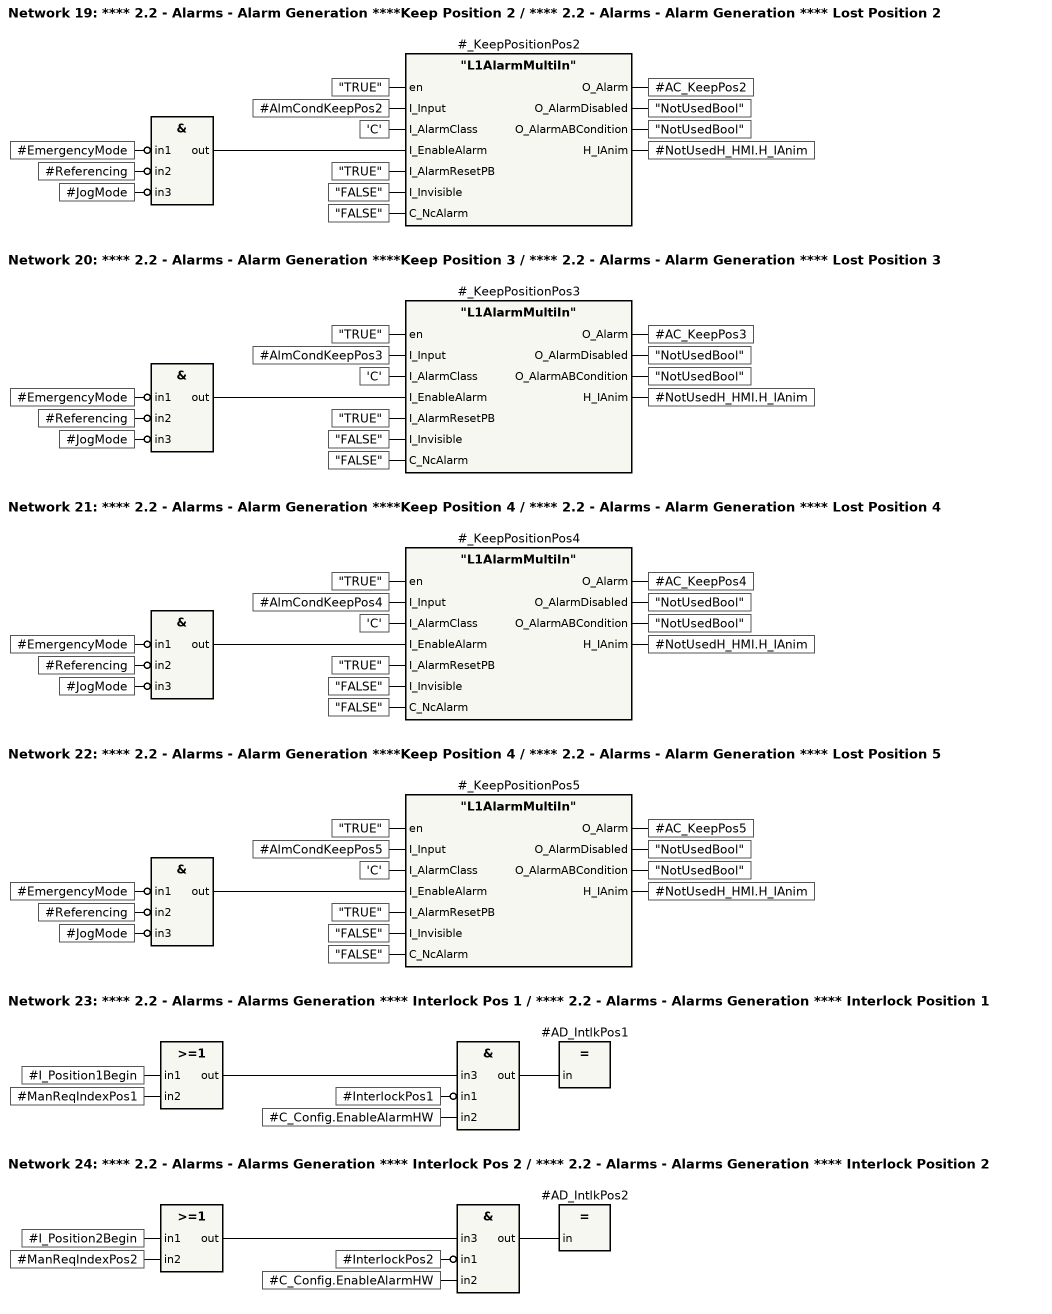
   IF "TRUE" THEN
       #_KeepPositionPos2(I_Input := #AlmCondKeepPos2,   // "L1AlarmMultiIn"
                          I_AlarmClass := 'C',
                          I_EnableAlarm := NOT #EmergencyMode AND NOT #Referencing AND NOT #JogMode,
                          I_AlarmResetPB := "TRUE",
                          I_Invisible := "FALSE",
                          C_NcAlarm := "FALSE",
                          O_Alarm => #AC_KeepPos2,
                          O_AlarmDisabled => "NotUsedBool",
                          O_AlarmABCondition => "NotUsedBool",
                          H_IAnim => #NotUsedH_HMI.H_IAnim);
   END_IF;
END_REGION

REGION Network 20: **** 2.2 - Alarms - Alarm Generation ****Keep Position 3 / **** 2.2 - Alarms - Alarm Generation **** Lost Position 3
   // Keep Position 3
   IF "TRUE" THEN
       #_KeepPositionPos3(I_Input := #AlmCondKeepPos3,   // "L1AlarmMultiIn"
                          I_AlarmClass := 'C',
                          I_EnableAlarm := NOT #EmergencyMode AND NOT #Referencing AND NOT #JogMode,
                          I_AlarmResetPB := "TRUE",
                          I_Invisible := "FALSE",
                          C_NcAlarm := "FALSE",
                          O_Alarm => #AC_KeepPos3,
                          O_AlarmDisabled => "NotUsedBool",
                          O_AlarmABCondition => "NotUsedBool",
                          H_IAnim => #NotUsedH_HMI.H_IAnim);
   END_IF;
END_REGION

REGION Network 21: **** 2.2 - Alarms - Alarm Generation ****Keep Position 4 / **** 2.2 - Alarms - Alarm Generation **** Lost Position 4
   // Keep Position 4
   IF "TRUE" THEN
       #_KeepPositionPos4(I_Input := #AlmCondKeepPos4,   // "L1AlarmMultiIn"
                          I_AlarmClass := 'C',
                          I_EnableAlarm := NOT #EmergencyMode AND NOT #Referencing AND NOT #JogMode,
                          I_AlarmResetPB := "TRUE",
                          I_Invisible := "FALSE",
                          C_NcAlarm := "FALSE",
                          O_Alarm => #AC_KeepPos4,
                          O_AlarmDisabled => "NotUsedBool",
                          O_AlarmABCondition => "NotUsedBool",
                          H_IAnim => #NotUsedH_HMI.H_IAnim);
   END_IF;
END_REGION

REGION Network 22: **** 2.2 - Alarms - Alarm Generation ****Keep Position 4 / **** 2.2 - Alarms - Alarm Generation **** Lost Position 5
   // Keep Position 4
   IF "TRUE" THEN
       #_KeepPositionPos5(I_Input := #AlmCondKeepPos5,   // "L1AlarmMultiIn"
                          I_AlarmClass := 'C',
                          I_EnableAlarm := NOT #EmergencyMode AND NOT #Referencing AND NOT #JogMode,
                          I_AlarmResetPB := "TRUE",
                          I_Invisible := "FALSE",
                          C_NcAlarm := "FALSE",
                          O_Alarm => #AC_KeepPos5,
                          O_AlarmDisabled => "NotUsedBool",
                          O_AlarmABCondition => "NotUsedBool",
                          H_IAnim => #NotUsedH_HMI.H_IAnim);
   END_IF;
END_REGION

REGION Network 23: **** 2.2 - Alarms - Alarms Generation **** Interlock Pos 1 / **** 2.2 - Alarms - Alarms Generation **** Interlock Position 1
   // Interlock Pos 1
   #AD_IntlkPos1 := (#I_Position1Begin OR #ManReqIndexPos1) AND NOT #InterlockPos1 AND #C_Config.EnableAlarmHW;
END_REGION

REGION Network 24: **** 2.2 - Alarms - Alarms Generation **** Interlock Pos 2 / **** 2.2 - Alarms - Alarms Generation **** Interlock Position 2
   // Interlock Pos 2
   #AD_IntlkPos2 := (#I_Position2Begin OR #ManReqIndexPos2) AND NOT #InterlockPos2 AND #C_Config.EnableAlarmHW;
END_REGION

REGION Network 25: **** 2.2 - Alarms - Alarms Generation **** Interlock Pos 3 / **** 2.2 - Alarms - Alarms Generation **** Interlock Position 3
   // Interlock Pos 3
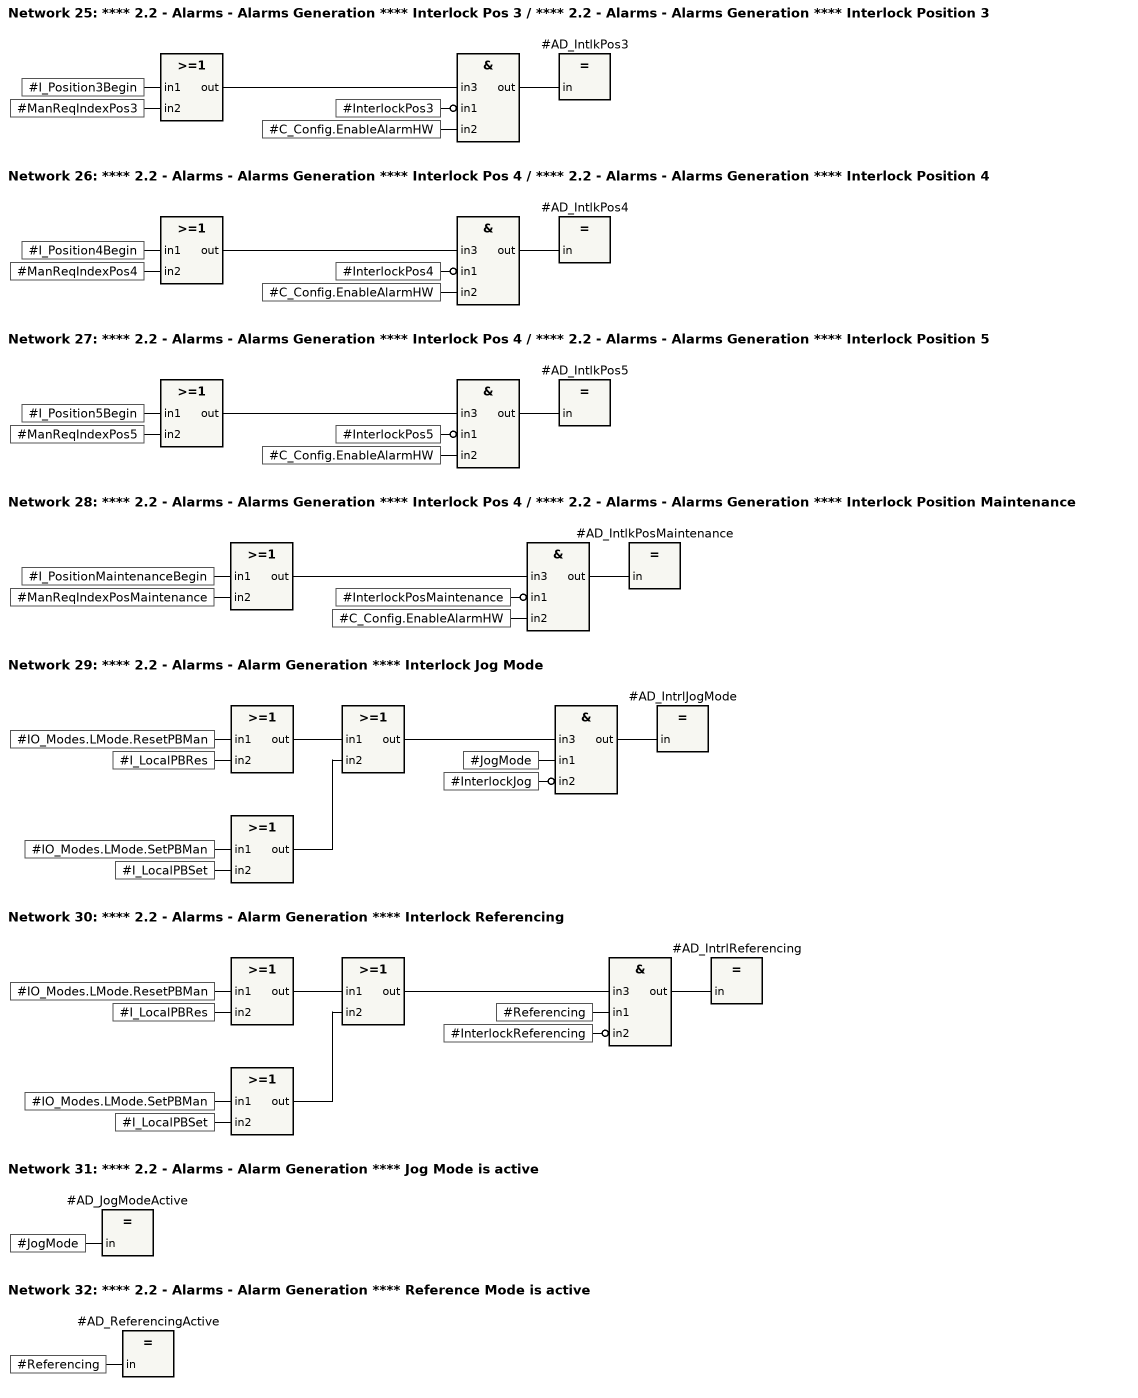
   #AD_IntlkPos3 := (#I_Position3Begin OR #ManReqIndexPos3) AND NOT #InterlockPos3 AND #C_Config.EnableAlarmHW;
END_REGION

REGION Network 26: **** 2.2 - Alarms - Alarms Generation **** Interlock Pos 4 / **** 2.2 - Alarms - Alarms Generation **** Interlock Position 4
   // Interlock Pos 4
   #AD_IntlkPos4 := (#I_Position4Begin OR #ManReqIndexPos4) AND NOT #InterlockPos4 AND #C_Config.EnableAlarmHW;
END_REGION

REGION Network 27: **** 2.2 - Alarms - Alarms Generation **** Interlock Pos 4 / **** 2.2 - Alarms - Alarms Generation **** Interlock Position 5
   // Interlock Pos 4
   #AD_IntlkPos5 := (#I_Position5Begin OR #ManReqIndexPos5) AND NOT #InterlockPos5 AND #C_Config.EnableAlarmHW;
END_REGION

REGION Network 28: **** 2.2 - Alarms - Alarms Generation **** Interlock Pos 4 / **** 2.2 - Alarms - Alarms Generation **** Interlock Position Maintenance
   // Interlock Pos 4
   #AD_IntlkPosMaintenance := (#I_PositionMaintenanceBegin OR #ManReqIndexPosMaintenance) AND NOT #InterlockPosMaintenance AND #C_Config.EnableAlarmHW;
END_REGION

REGION Network 29: **** 2.2 - Alarms - Alarm Generation **** Interlock Jog Mode
   #AD_IntrlJogMode := (#IO_Modes.LMode.ResetPBMan OR #I_LocalPBRes OR #IO_Modes.LMode.SetPBMan OR #I_LocalPBSet) AND #JogMode AND NOT #InterlockJog;
END_REGION

REGION Network 30: **** 2.2 - Alarms - Alarm Generation **** Interlock Referencing
   #AD_IntrlReferencing := (#IO_Modes.LMode.ResetPBMan OR #I_LocalPBRes OR #IO_Modes.LMode.SetPBMan OR #I_LocalPBSet) AND #Referencing AND NOT #InterlockReferencing;
END_REGION

REGION Network 31: **** 2.2 - Alarms - Alarm Generation **** Jog Mode is active
   #AD_JogModeActive := #JogMode;
END_REGION

REGION Network 32: **** 2.2 - Alarms - Alarm Generation **** Reference Mode is active
   #AD_ReferencingActive := #Referencing;
END_REGION

REGION Network 33: **** 2.2 - Alarms - Alarm Generation **** Emergency Mode is active
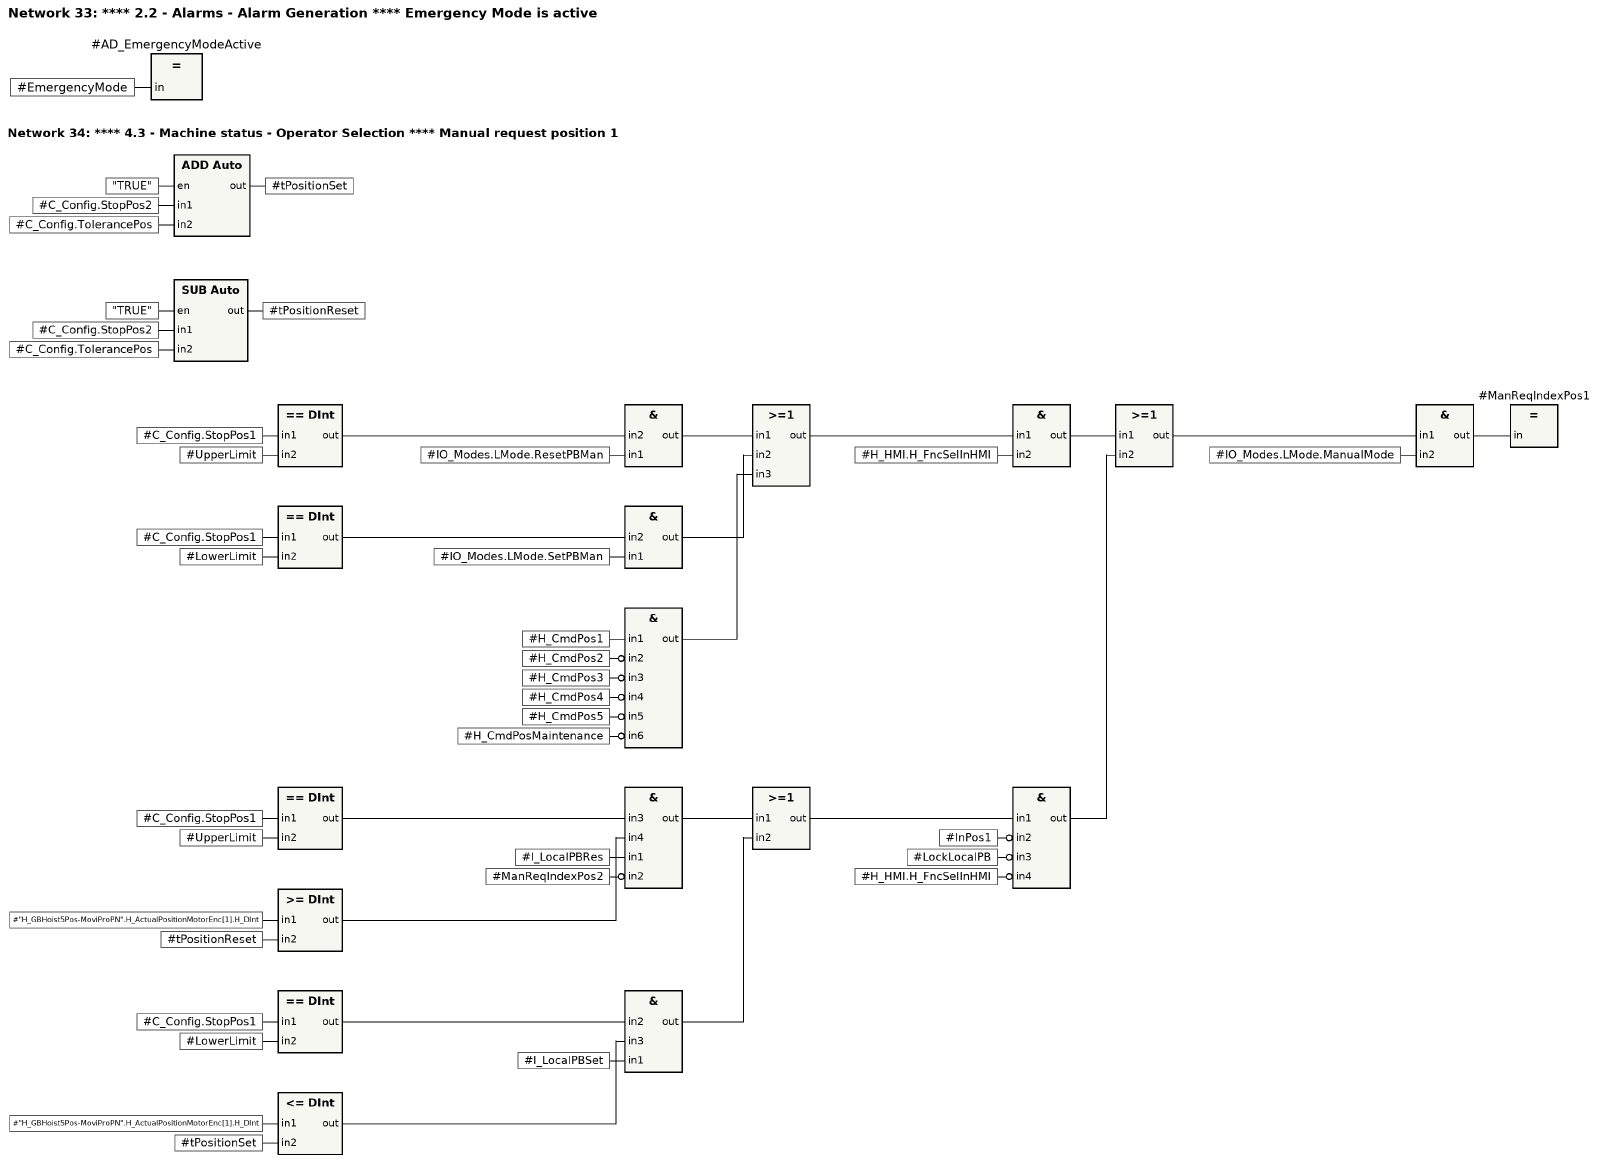
   #AD_EmergencyModeActive := #EmergencyMode;
END_REGION

REGION Network 34: **** 4.3 - Machine status - Operator Selection **** Manual request position 1
   IF "TRUE" THEN
       #tPositionSet := #C_Config.StopPos2 + #C_Config.TolerancePos;
       #tPositionReset := #C_Config.StopPos2 - #C_Config.TolerancePos;
   END_IF;
   #ManReqIndexPos1 := (((((#C_Config.StopPos1 = #UpperLimit) AND #IO_Modes.LMode.ResetPBMan) OR ((#C_Config.StopPos1 = #LowerLimit) AND #IO_Modes.LMode.SetPBMan) OR (#H_CmdPos1 AND NOT #H_CmdPos2 AND NOT #H_CmdPos3 AND NOT #H_CmdPos4 AND NOT #H_CmdPos5 AND NOT #H_CmdPosMaintenance)) AND #H_HMI.H_FncSelInHMI) OR ((((#C_Config.StopPos1 = #UpperLimit) AND (#"H_GBHoist5Pos-MoviProPN".H_ActualPositionMotorEnc[1].H_DInt >= #tPositionReset) AND #I_LocalPBRes AND NOT #ManReqIndexPos2) OR ((#C_Config.StopPos1 = #LowerLimit) AND (#"H_GBHoist5Pos-MoviProPN".H_ActualPositionMotorEnc[1].H_DInt <= #tPositionSet) AND #I_LocalPBSet)) AND NOT #InPos1 AND NOT #LockLocalPB AND NOT #H_HMI.H_FncSelInHMI)) AND #IO_Modes.LMode.ManualMode;
END_REGION

REGION Network 35: **** 4.3 - Machine status - Operator Selection **** Manual request position 2
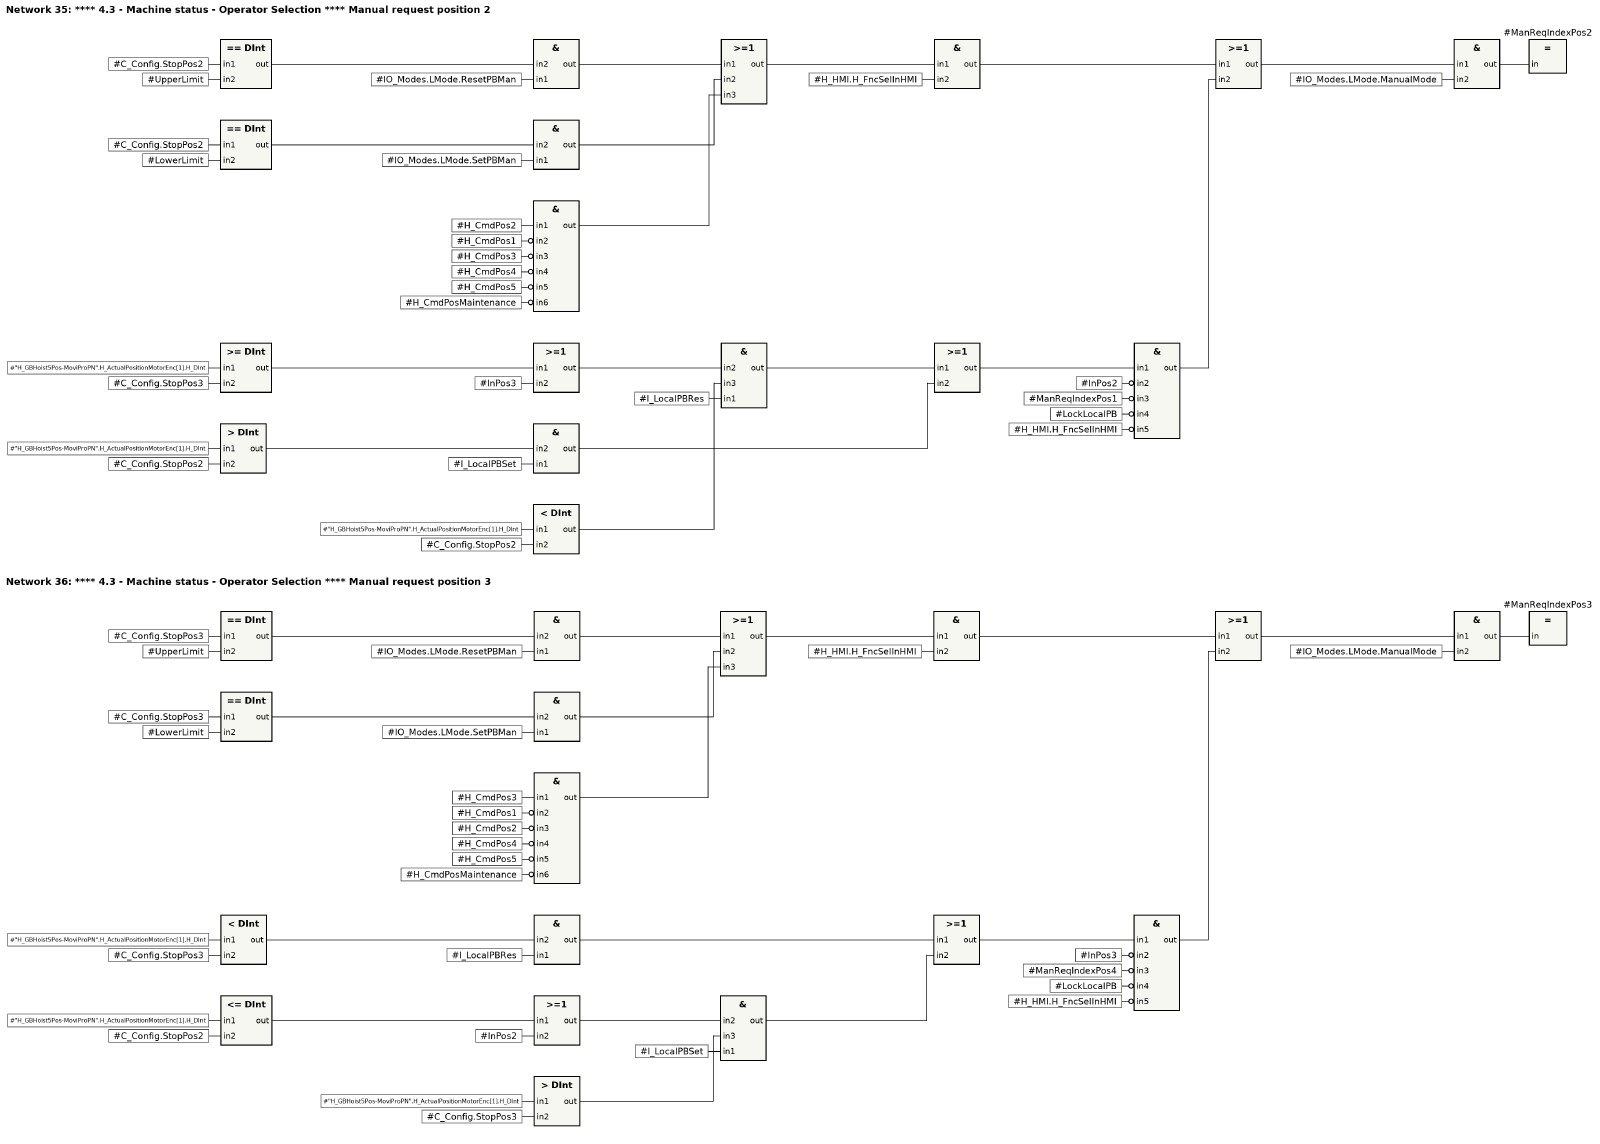
   #ManReqIndexPos2 := (((((#C_Config.StopPos2 = #UpperLimit) AND #IO_Modes.LMode.ResetPBMan) OR ((#C_Config.StopPos2 = #LowerLimit) AND #IO_Modes.LMode.SetPBMan) OR (#H_CmdPos2 AND NOT #H_CmdPos1 AND NOT #H_CmdPos3 AND NOT #H_CmdPos4 AND NOT #H_CmdPos5 AND NOT #H_CmdPosMaintenance)) AND #H_HMI.H_FncSelInHMI) OR (((((#"H_GBHoist5Pos-MoviProPN".H_ActualPositionMotorEnc[1].H_DInt >= #C_Config.StopPos3) OR #InPos3) AND (#"H_GBHoist5Pos-MoviProPN".H_ActualPositionMotorEnc[1].H_DInt < #C_Config.StopPos2) AND #I_LocalPBRes) OR ((#"H_GBHoist5Pos-MoviProPN".H_ActualPositionMotorEnc[1].H_DInt > #C_Config.StopPos2) AND #I_LocalPBSet)) AND NOT #InPos2 AND NOT #ManReqIndexPos1 AND NOT #LockLocalPB AND NOT #H_HMI.H_FncSelInHMI)) AND #IO_Modes.LMode.ManualMode;
END_REGION

REGION Network 36: **** 4.3 - Machine status - Operator Selection **** Manual request position 3
   #ManReqIndexPos3 := (((((#C_Config.StopPos3 = #UpperLimit) AND #IO_Modes.LMode.ResetPBMan) OR ((#C_Config.StopPos3 = #LowerLimit) AND #IO_Modes.LMode.SetPBMan) OR (#H_CmdPos3 AND NOT #H_CmdPos1 AND NOT #H_CmdPos2 AND NOT #H_CmdPos4 AND NOT #H_CmdPos5 AND NOT #H_CmdPosMaintenance)) AND #H_HMI.H_FncSelInHMI) OR ((((#"H_GBHoist5Pos-MoviProPN".H_ActualPositionMotorEnc[1].H_DInt < #C_Config.StopPos3) AND #I_LocalPBRes) OR (((#"H_GBHoist5Pos-MoviProPN".H_ActualPositionMotorEnc[1].H_DInt <= #C_Config.StopPos2) OR #InPos2) AND (#"H_GBHoist5Pos-MoviProPN".H_ActualPositionMotorEnc[1].H_DInt > #C_Config.StopPos3) AND #I_LocalPBSet)) AND NOT #InPos3 AND NOT #ManReqIndexPos4 AND NOT #LockLocalPB AND NOT #H_HMI.H_FncSelInHMI)) AND #IO_Modes.LMode.ManualMode;
END_REGION

REGION Network 37: **** 4.3 - Machine status - Operator Selection **** Manual request position 3 / **** 4.3 - Machine status - Operator Selection **** Manual request position 4
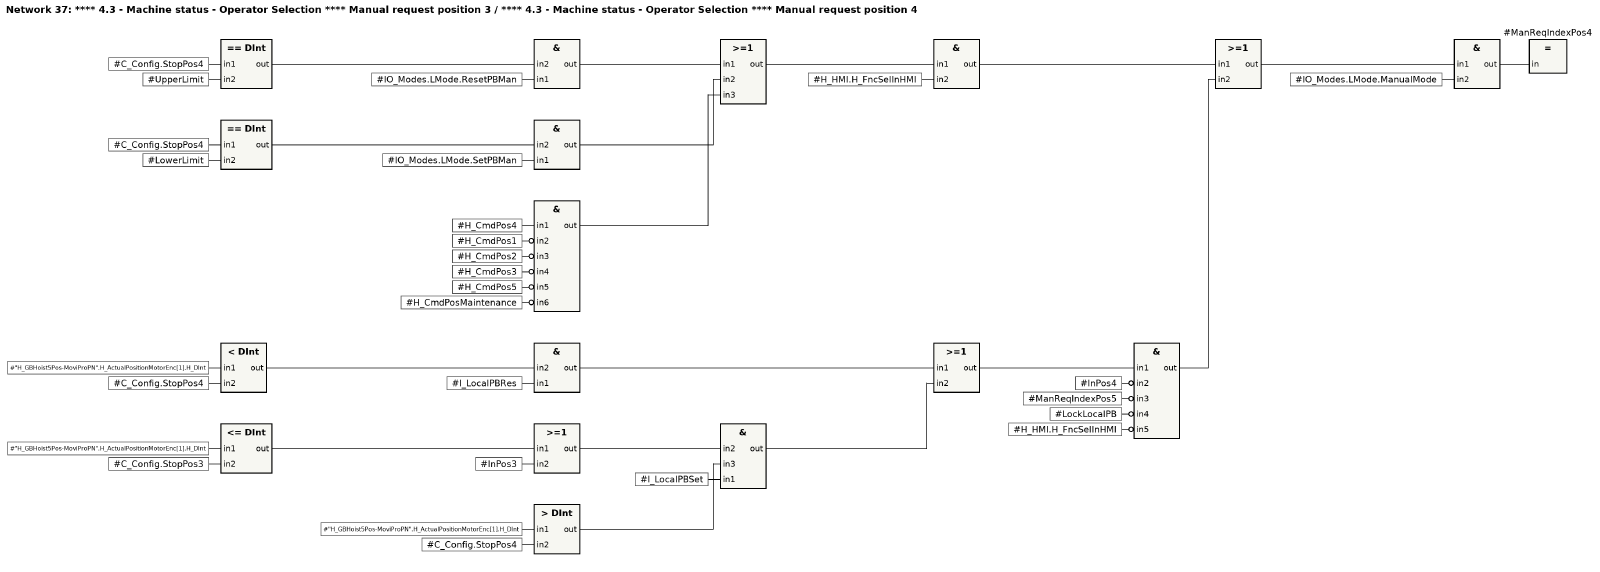
   #ManReqIndexPos4 := (((((#C_Config.StopPos4 = #UpperLimit) AND #IO_Modes.LMode.ResetPBMan) OR ((#C_Config.StopPos4 = #LowerLimit) AND #IO_Modes.LMode.SetPBMan) OR (#H_CmdPos4 AND NOT #H_CmdPos1 AND NOT #H_CmdPos2 AND NOT #H_CmdPos3 AND NOT #H_CmdPos5 AND NOT #H_CmdPosMaintenance)) AND #H_HMI.H_FncSelInHMI) OR ((((#"H_GBHoist5Pos-MoviProPN".H_ActualPositionMotorEnc[1].H_DInt < #C_Config.StopPos4) AND #I_LocalPBRes) OR (((#"H_GBHoist5Pos-MoviProPN".H_ActualPositionMotorEnc[1].H_DInt <= #C_Config.StopPos3) OR #InPos3) AND (#"H_GBHoist5Pos-MoviProPN".H_ActualPositionMotorEnc[1].H_DInt > #C_Config.StopPos4) AND #I_LocalPBSet)) AND NOT #InPos4 AND NOT #ManReqIndexPos5 AND NOT #LockLocalPB AND NOT #H_HMI.H_FncSelInHMI)) AND #IO_Modes.LMode.ManualMode;
END_REGION

REGION Network 38: **** 4.3 - Machine status - Operator Selection **** Manual request position 4 / **** 4.3 - Machine status - Operator Selection **** Manual request position 5
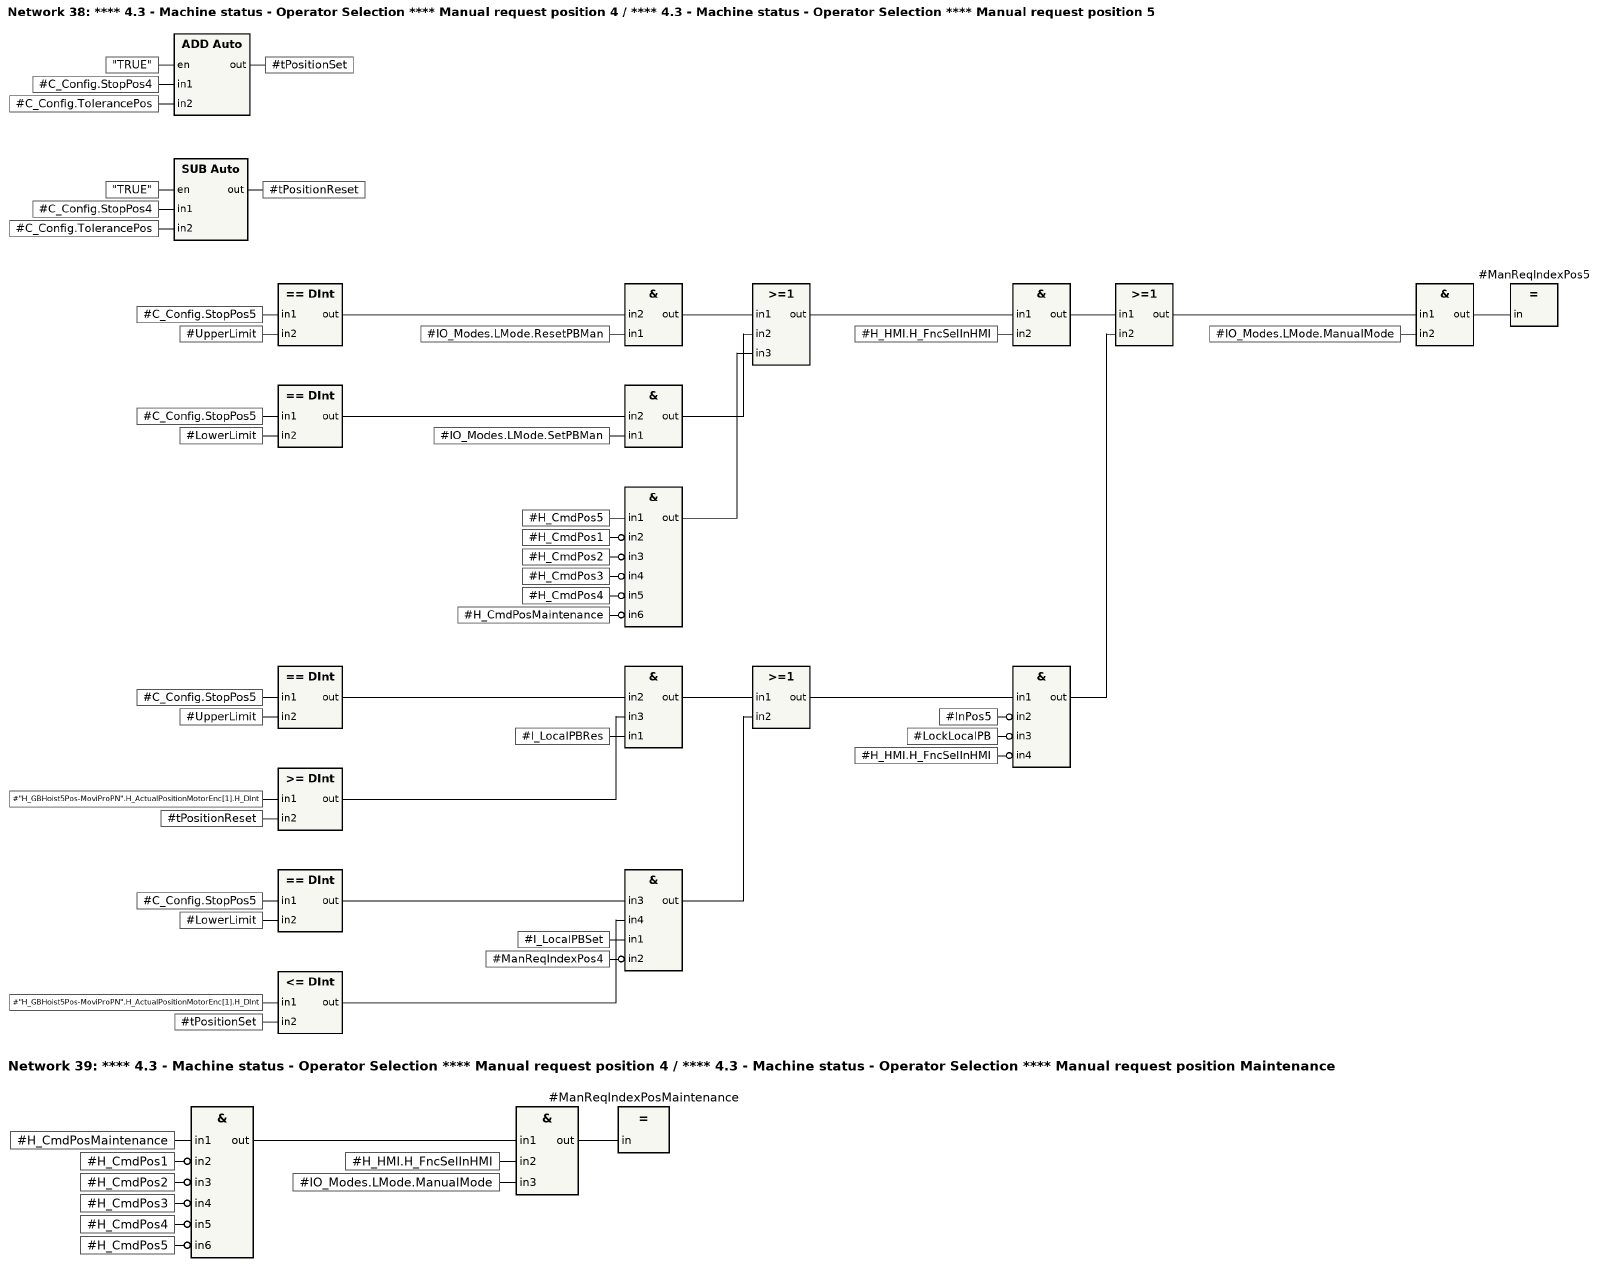
   IF "TRUE" THEN
       #tPositionSet := #C_Config.StopPos4 + #C_Config.TolerancePos;
       #tPositionReset := #C_Config.StopPos4 - #C_Config.TolerancePos;
   END_IF;
   #ManReqIndexPos5 := (((((#C_Config.StopPos5 = #UpperLimit) AND #IO_Modes.LMode.ResetPBMan) OR ((#C_Config.StopPos5 = #LowerLimit) AND #IO_Modes.LMode.SetPBMan) OR (#H_CmdPos5 AND NOT #H_CmdPos1 AND NOT #H_CmdPos2 AND NOT #H_CmdPos3 AND NOT #H_CmdPos4 AND NOT #H_CmdPosMaintenance)) AND #H_HMI.H_FncSelInHMI) OR ((((#C_Config.StopPos5 = #UpperLimit) AND (#"H_GBHoist5Pos-MoviProPN".H_ActualPositionMotorEnc[1].H_DInt >= #tPositionReset) AND #I_LocalPBRes) OR ((#C_Config.StopPos5 = #LowerLimit) AND (#"H_GBHoist5Pos-MoviProPN".H_ActualPositionMotorEnc[1].H_DInt <= #tPositionSet) AND #I_LocalPBSet AND NOT #ManReqIndexPos4)) AND NOT #InPos5 AND NOT #LockLocalPB AND NOT #H_HMI.H_FncSelInHMI)) AND #IO_Modes.LMode.ManualMode;
END_REGION

REGION Network 39: **** 4.3 - Machine status - Operator Selection **** Manual request position 4 / **** 4.3 - Machine status - Operator Selection **** Manual request position Maintenance
   #ManReqIndexPosMaintenance := #H_CmdPosMaintenance AND NOT #H_CmdPos1 AND NOT #H_CmdPos2 AND NOT #H_CmdPos3 AND NOT #H_CmdPos4 AND NOT #H_CmdPos5 AND #H_HMI.H_FncSelInHMI AND #IO_Modes.LMode.ManualMode;
END_REGION

REGION Network 40: **** 4.3 - Machine status - Operator Selection **** Reset H_SelInHMI
   // Reset H_SelInHMI
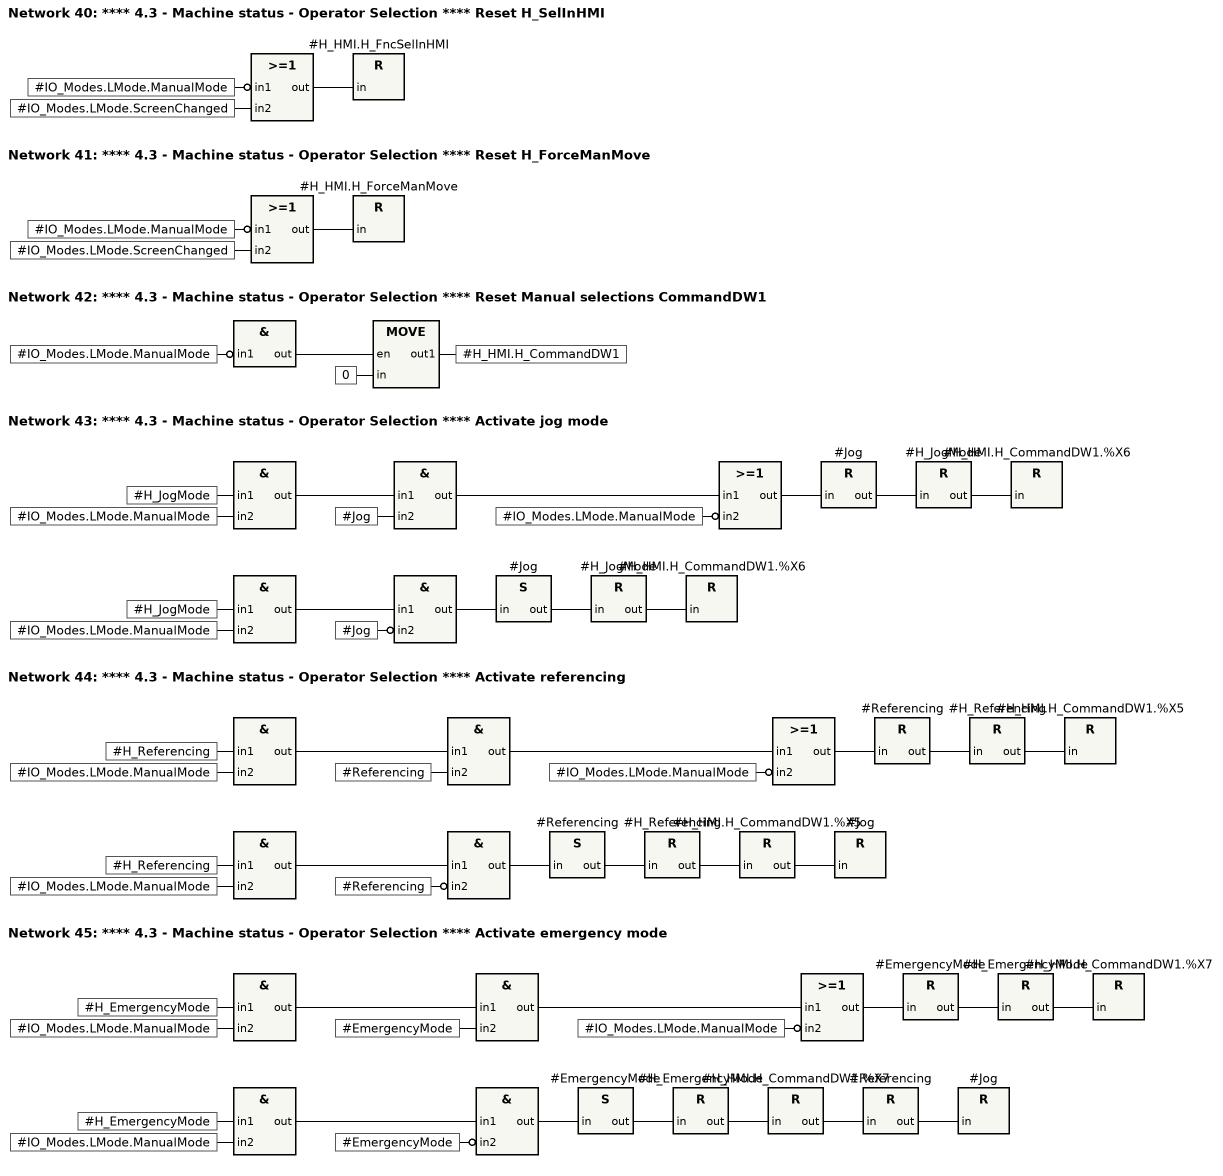
   IF NOT #IO_Modes.LMode.ManualMode OR #IO_Modes.LMode.ScreenChanged THEN
       #H_HMI.H_FncSelInHMI := FALSE;
   END_IF;
END_REGION

REGION Network 41: **** 4.3 - Machine status - Operator Selection **** Reset H_ForceManMove
   // Reset H_ForceManMove
   IF NOT #IO_Modes.LMode.ManualMode OR #IO_Modes.LMode.ScreenChanged THEN
       #H_HMI.H_ForceManMove := FALSE;
   END_IF;
END_REGION

REGION Network 42: **** 4.3 - Machine status - Operator Selection **** Reset Manual selections CommandDW1
   // Reset all selections in the HMI
   IF NOT #IO_Modes.LMode.ManualMode THEN #H_HMI.H_CommandDW1 := 0; END_IF;
END_REGION

REGION Network 43: **** 4.3 - Machine status - Operator Selection **** Activate jog mode
   // Reset H_ForceManMove
   #_w1 := (#H_JogMode AND #IO_Modes.LMode.ManualMode AND #Jog) OR NOT #IO_Modes.LMode.ManualMode;
   IF #_w1 THEN
       #Jog := FALSE;
       #H_JogMode := FALSE;
       #H_HMI.H_CommandDW1.%X6 := FALSE;
   END_IF;
   #_w2 := #H_JogMode AND #IO_Modes.LMode.ManualMode AND NOT #Jog;
   IF #_w2 THEN
       #Jog := TRUE;
       #H_JogMode := FALSE;
       #H_HMI.H_CommandDW1.%X6 := FALSE;
   END_IF;
END_REGION

REGION Network 44: **** 4.3 - Machine status - Operator Selection **** Activate referencing
   // Calibration procedure initiated from HMI panel
   #_w1 := (#H_Referencing AND #IO_Modes.LMode.ManualMode AND #Referencing) OR NOT #IO_Modes.LMode.ManualMode;
   IF #_w1 THEN
       #Referencing := FALSE;
       #H_Referencing := FALSE;
       #H_HMI.H_CommandDW1.%X5 := FALSE;
   END_IF;
   #_w2 := #H_Referencing AND #IO_Modes.LMode.ManualMode AND NOT #Referencing;
   IF #_w2 THEN
       #Referencing := TRUE;
       #H_Referencing := FALSE;
       #H_HMI.H_CommandDW1.%X5 := FALSE;
       #Jog := FALSE;
   END_IF;
END_REGION

REGION Network 45: **** 4.3 - Machine status - Operator Selection **** Activate emergency mode
   // Activate emergency mode
   #_w1 := (#H_EmergencyMode AND #IO_Modes.LMode.ManualMode AND #EmergencyMode) OR NOT #IO_Modes.LMode.ManualMode;
   IF #_w1 THEN
       #EmergencyMode := FALSE;
       #H_EmergencyMode := FALSE;
       #H_HMI.H_CommandDW1.%X7 := FALSE;
   END_IF;
   #_w2 := #H_EmergencyMode AND #IO_Modes.LMode.ManualMode AND NOT #EmergencyMode;
   IF #_w2 THEN
       #EmergencyMode := TRUE;
       #H_EmergencyMode := FALSE;
       #H_HMI.H_CommandDW1.%X7 := FALSE;
       #Referencing := FALSE;
       #Jog := FALSE;
   END_IF;
END_REGION

REGION Network 46: **** 4.4 - Machine status - Calculation **** Lower limit position
   // Calculate minimum value of all positions
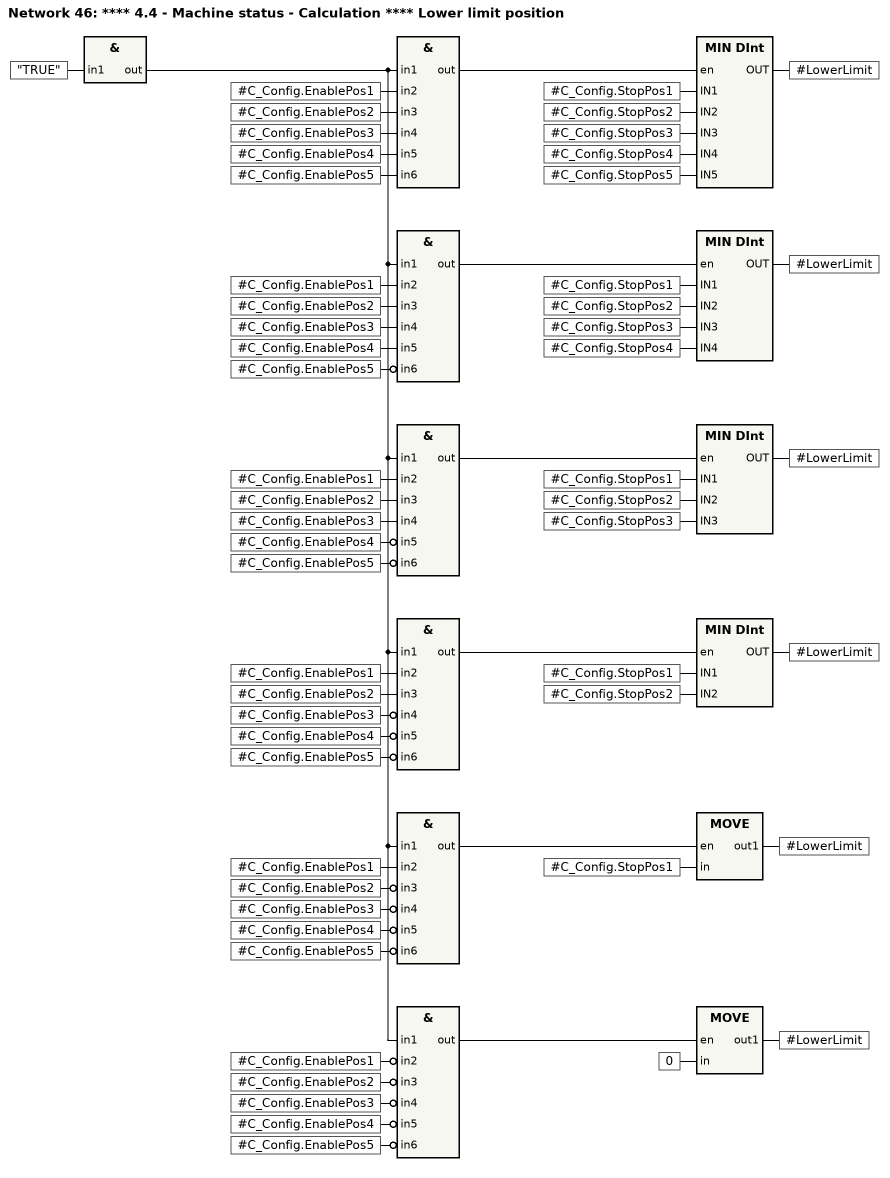
   IF "TRUE" AND #C_Config.EnablePos1 AND #C_Config.EnablePos2 AND #C_Config.EnablePos3 AND #C_Config.EnablePos4 AND #C_Config.EnablePos5 THEN
       #LowerLimit := MIN(IN1 := #C_Config.StopPos1, IN2 := #C_Config.StopPos2, IN3 := #C_Config.StopPos3, IN4 := #C_Config.StopPos4, IN5 := #C_Config.StopPos5);
   END_IF;
   IF "TRUE" AND #C_Config.EnablePos1 AND #C_Config.EnablePos2 AND #C_Config.EnablePos3 AND #C_Config.EnablePos4 AND NOT #C_Config.EnablePos5 THEN
       #LowerLimit := MIN(IN1 := #C_Config.StopPos1, IN2 := #C_Config.StopPos2, IN3 := #C_Config.StopPos3, IN4 := #C_Config.StopPos4);
   END_IF;
   IF "TRUE" AND #C_Config.EnablePos1 AND #C_Config.EnablePos2 AND #C_Config.EnablePos3 AND NOT #C_Config.EnablePos4 AND NOT #C_Config.EnablePos5 THEN
       #LowerLimit := MIN(IN1 := #C_Config.StopPos1, IN2 := #C_Config.StopPos2, IN3 := #C_Config.StopPos3);
   END_IF;
   IF "TRUE" AND #C_Config.EnablePos1 AND #C_Config.EnablePos2 AND NOT #C_Config.EnablePos3 AND NOT #C_Config.EnablePos4 AND NOT #C_Config.EnablePos5 THEN
       #LowerLimit := MIN(IN1 := #C_Config.StopPos1, IN2 := #C_Config.StopPos2);
   END_IF;
   IF "TRUE" AND #C_Config.EnablePos1 AND NOT #C_Config.EnablePos2 AND NOT #C_Config.EnablePos3 AND NOT #C_Config.EnablePos4 AND NOT #C_Config.EnablePos5 THEN
       #LowerLimit := #C_Config.StopPos1;
   END_IF;
   IF "TRUE" AND NOT #C_Config.EnablePos1 AND NOT #C_Config.EnablePos2 AND NOT #C_Config.EnablePos3 AND NOT #C_Config.EnablePos4 AND NOT #C_Config.EnablePos5 THEN
       #LowerLimit := 0;
   END_IF;
END_REGION

REGION Network 47: **** 4.4 - Machine status - Calculation **** Upper limit position
   // Calculate maximum value of all positions
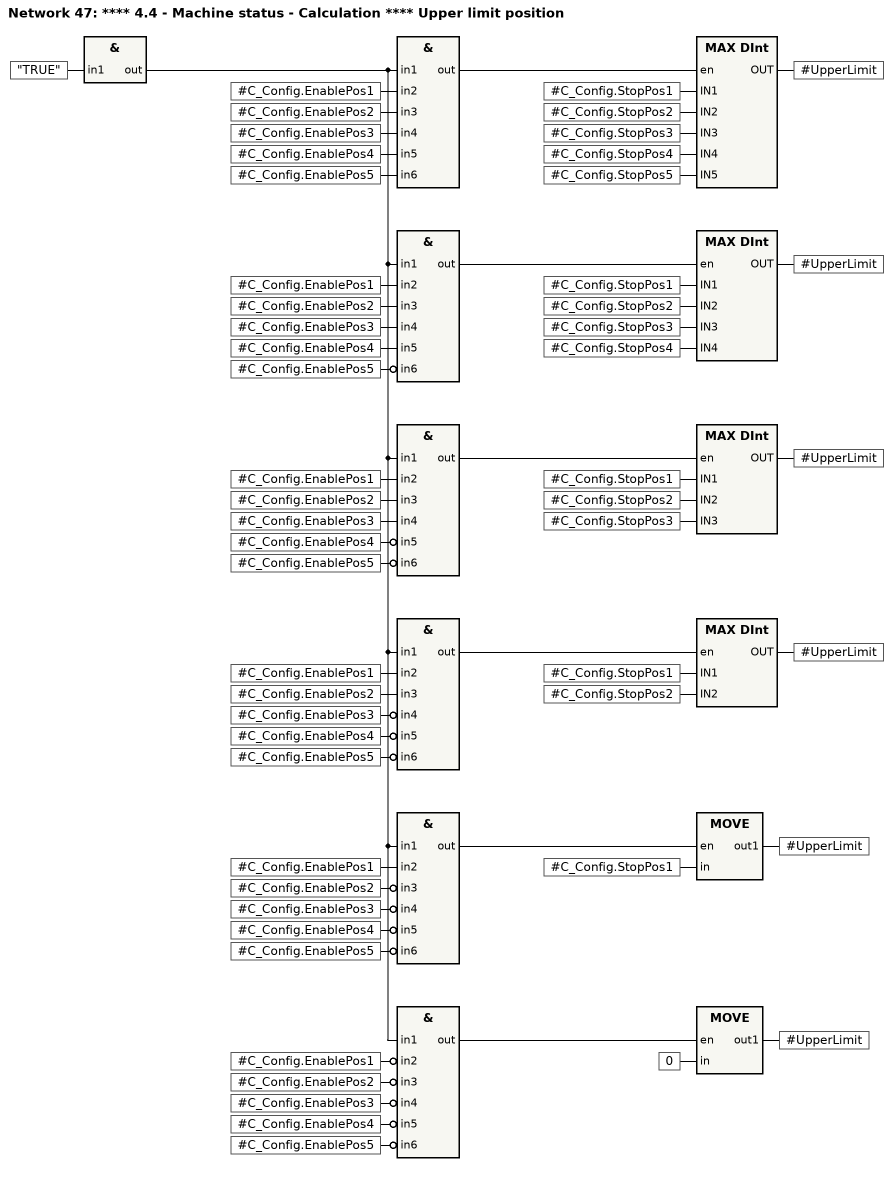
   IF "TRUE" AND #C_Config.EnablePos1 AND #C_Config.EnablePos2 AND #C_Config.EnablePos3 AND #C_Config.EnablePos4 AND #C_Config.EnablePos5 THEN
       #UpperLimit := MAX(IN1 := #C_Config.StopPos1, IN2 := #C_Config.StopPos2, IN3 := #C_Config.StopPos3, IN4 := #C_Config.StopPos4, IN5 := #C_Config.StopPos5);
   END_IF;
   IF "TRUE" AND #C_Config.EnablePos1 AND #C_Config.EnablePos2 AND #C_Config.EnablePos3 AND #C_Config.EnablePos4 AND NOT #C_Config.EnablePos5 THEN
       #UpperLimit := MAX(IN1 := #C_Config.StopPos1, IN2 := #C_Config.StopPos2, IN3 := #C_Config.StopPos3, IN4 := #C_Config.StopPos4);
   END_IF;
   IF "TRUE" AND #C_Config.EnablePos1 AND #C_Config.EnablePos2 AND #C_Config.EnablePos3 AND NOT #C_Config.EnablePos4 AND NOT #C_Config.EnablePos5 THEN
       #UpperLimit := MAX(IN1 := #C_Config.StopPos1, IN2 := #C_Config.StopPos2, IN3 := #C_Config.StopPos3);
   END_IF;
   IF "TRUE" AND #C_Config.EnablePos1 AND #C_Config.EnablePos2 AND NOT #C_Config.EnablePos3 AND NOT #C_Config.EnablePos4 AND NOT #C_Config.EnablePos5 THEN
       #UpperLimit := MAX(IN1 := #C_Config.StopPos1, IN2 := #C_Config.StopPos2);
   END_IF;
   IF "TRUE" AND #C_Config.EnablePos1 AND NOT #C_Config.EnablePos2 AND NOT #C_Config.EnablePos3 AND NOT #C_Config.EnablePos4 AND NOT #C_Config.EnablePos5 THEN
       #UpperLimit := #C_Config.StopPos1;
   END_IF;
   IF "TRUE" AND NOT #C_Config.EnablePos1 AND NOT #C_Config.EnablePos2 AND NOT #C_Config.EnablePos3 AND NOT #C_Config.EnablePos4 AND NOT #C_Config.EnablePos5 THEN
       #UpperLimit := 0;
   END_IF;
END_REGION

REGION Network 48: **** 4.6 - Machine Status - Indication **** Stop Detection High Speed Set / **** 4.6 - Machine Status - Indication **** Belt check sensor 1
   // Stop Detection High Speed Set
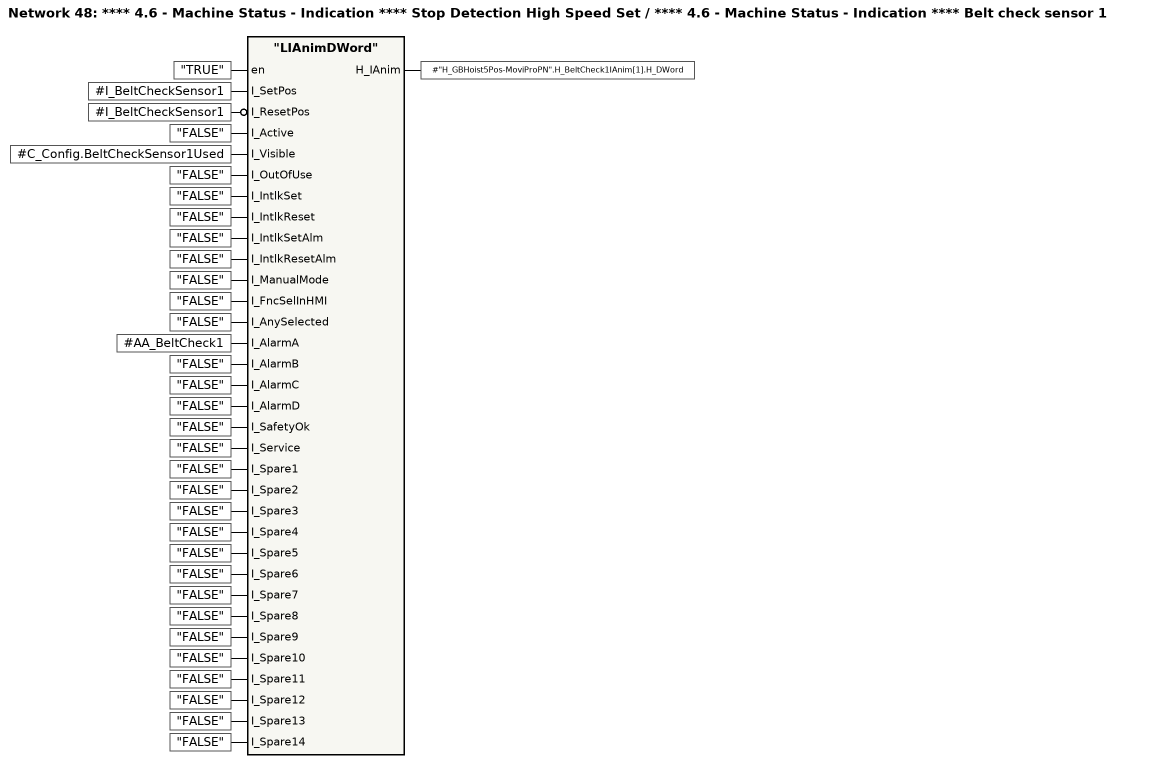
   IF "TRUE" THEN
       "LIAnimDWord"(I_SetPos := #I_BeltCheckSensor1,
                     I_ResetPos := NOT #I_BeltCheckSensor1,
                     I_Active := "FALSE",
                     I_Visible := #C_Config.BeltCheckSensor1Used,
                     I_OutOfUse := "FALSE",
                     I_IntlkSet := "FALSE",
                     I_IntlkReset := "FALSE",
                     I_IntlkSetAlm := "FALSE",
                     I_IntlkResetAlm := "FALSE",
                     I_ManualMode := "FALSE",
                     I_FncSelInHMI := "FALSE",
                     I_AnySelected := "FALSE",
                     I_AlarmA := #AA_BeltCheck1,
                     I_AlarmB := "FALSE",
                     I_AlarmC := "FALSE",
                     I_AlarmD := "FALSE",
                     I_SafetyOk := "FALSE",
                     I_Service := "FALSE",
                     I_Spare1 := "FALSE",
                     I_Spare2 := "FALSE",
                     I_Spare3 := "FALSE",
                     I_Spare4 := "FALSE",
                     I_Spare5 := "FALSE",
                     I_Spare6 := "FALSE",
                     I_Spare7 := "FALSE",
                     I_Spare8 := "FALSE",
                     I_Spare9 := "FALSE",
                     I_Spare10 := "FALSE",
                     I_Spare11 := "FALSE",
                     I_Spare12 := "FALSE",
                     I_Spare13 := "FALSE",
                     I_Spare14 := "FALSE",
                     H_IAnim => #"H_GBHoist5Pos-MoviProPN".H_BeltCheck1IAnim[1].H_DWord);
   END_IF;
END_REGION

REGION Network 49: **** 4.6 - Machine Status - Indication **** Stop Detection High Speed Set / **** 4.6 - Machine Status - Indication **** Belt check sensor 2
   // Stop Detection High Speed Set
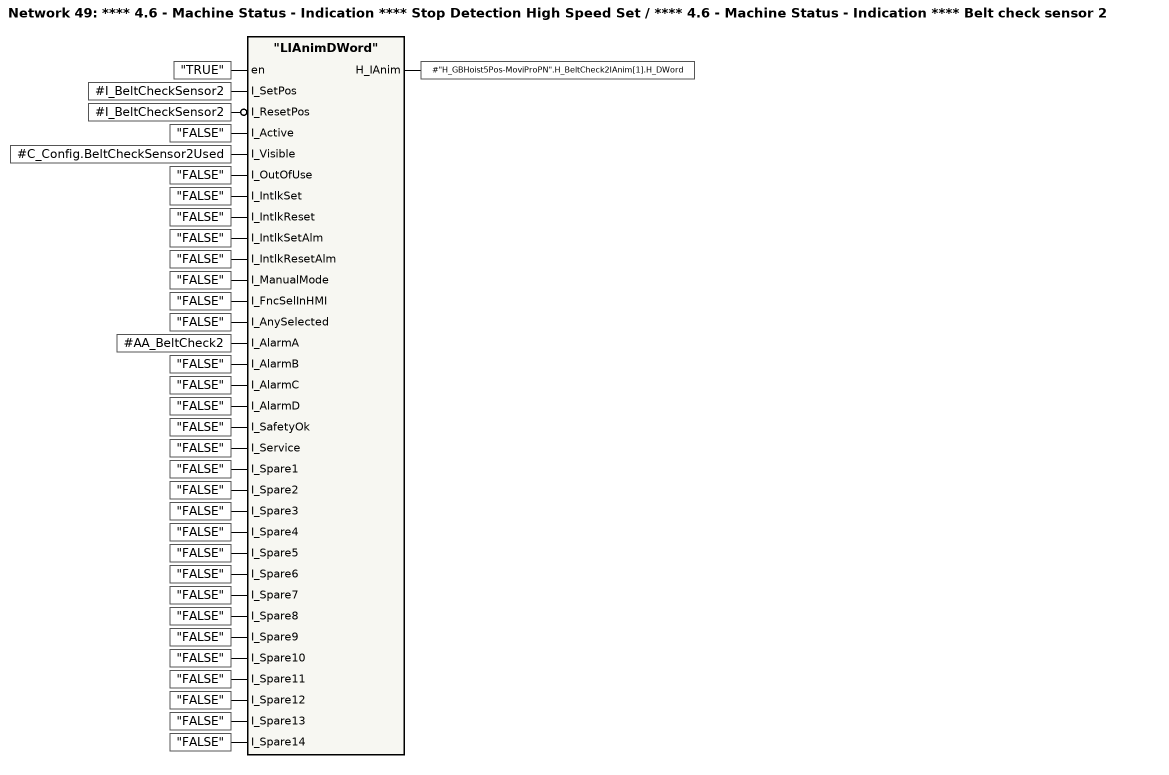
   IF "TRUE" THEN
       "LIAnimDWord"(I_SetPos := #I_BeltCheckSensor2,
                     I_ResetPos := NOT #I_BeltCheckSensor2,
                     I_Active := "FALSE",
                     I_Visible := #C_Config.BeltCheckSensor2Used,
                     I_OutOfUse := "FALSE",
                     I_IntlkSet := "FALSE",
                     I_IntlkReset := "FALSE",
                     I_IntlkSetAlm := "FALSE",
                     I_IntlkResetAlm := "FALSE",
                     I_ManualMode := "FALSE",
                     I_FncSelInHMI := "FALSE",
                     I_AnySelected := "FALSE",
                     I_AlarmA := #AA_BeltCheck2,
                     I_AlarmB := "FALSE",
                     I_AlarmC := "FALSE",
                     I_AlarmD := "FALSE",
                     I_SafetyOk := "FALSE",
                     I_Service := "FALSE",
                     I_Spare1 := "FALSE",
                     I_Spare2 := "FALSE",
                     I_Spare3 := "FALSE",
                     I_Spare4 := "FALSE",
                     I_Spare5 := "FALSE",
                     I_Spare6 := "FALSE",
                     I_Spare7 := "FALSE",
                     I_Spare8 := "FALSE",
                     I_Spare9 := "FALSE",
                     I_Spare10 := "FALSE",
                     I_Spare11 := "FALSE",
                     I_Spare12 := "FALSE",
                     I_Spare13 := "FALSE",
                     I_Spare14 := "FALSE",
                     H_IAnim => #"H_GBHoist5Pos-MoviProPN".H_BeltCheck2IAnim[1].H_DWord);
   END_IF;
END_REGION

REGION Network 50: **** 4.6 - Machine Status - Indication **** Stop Detection High Speed Set / **** 4.6 - Machine Status - Indication **** Clutch detection 1
   // Stop Detection High Speed Set
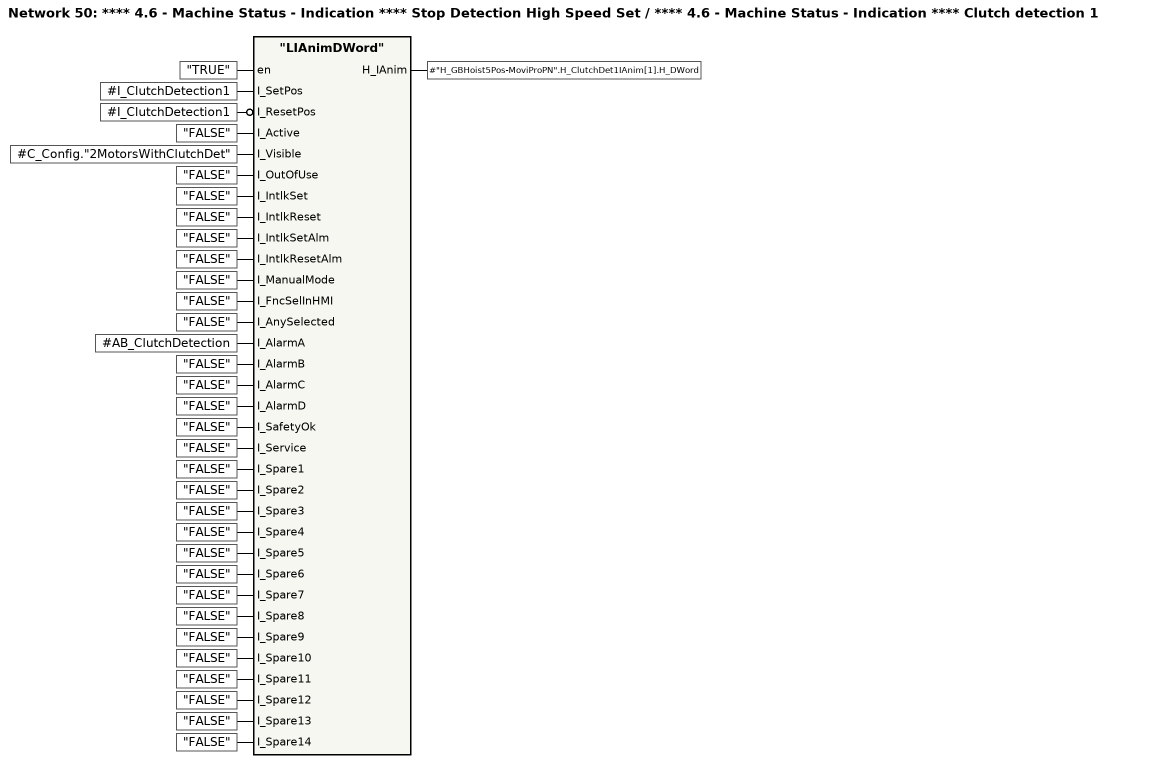
   IF "TRUE" THEN
       "LIAnimDWord"(I_SetPos := #I_ClutchDetection1,
                     I_ResetPos := NOT #I_ClutchDetection1,
                     I_Active := "FALSE",
                     I_Visible := #C_Config."2MotorsWithClutchDet",
                     I_OutOfUse := "FALSE",
                     I_IntlkSet := "FALSE",
                     I_IntlkReset := "FALSE",
                     I_IntlkSetAlm := "FALSE",
                     I_IntlkResetAlm := "FALSE",
                     I_ManualMode := "FALSE",
                     I_FncSelInHMI := "FALSE",
                     I_AnySelected := "FALSE",
                     I_AlarmA := #AB_ClutchDetection,
                     I_AlarmB := "FALSE",
                     I_AlarmC := "FALSE",
                     I_AlarmD := "FALSE",
                     I_SafetyOk := "FALSE",
                     I_Service := "FALSE",
                     I_Spare1 := "FALSE",
                     I_Spare2 := "FALSE",
                     I_Spare3 := "FALSE",
                     I_Spare4 := "FALSE",
                     I_Spare5 := "FALSE",
                     I_Spare6 := "FALSE",
                     I_Spare7 := "FALSE",
                     I_Spare8 := "FALSE",
                     I_Spare9 := "FALSE",
                     I_Spare10 := "FALSE",
                     I_Spare11 := "FALSE",
                     I_Spare12 := "FALSE",
                     I_Spare13 := "FALSE",
                     I_Spare14 := "FALSE",
                     H_IAnim => #"H_GBHoist5Pos-MoviProPN".H_ClutchDet1IAnim[1].H_DWord);
   END_IF;
END_REGION

REGION Network 51: **** 4.6 - Machine Status - Indication **** Stop Detection High Speed Set / **** 4.6 - Machine Status - Indication **** Clutch detection 2
   // Stop Detection High Speed Set
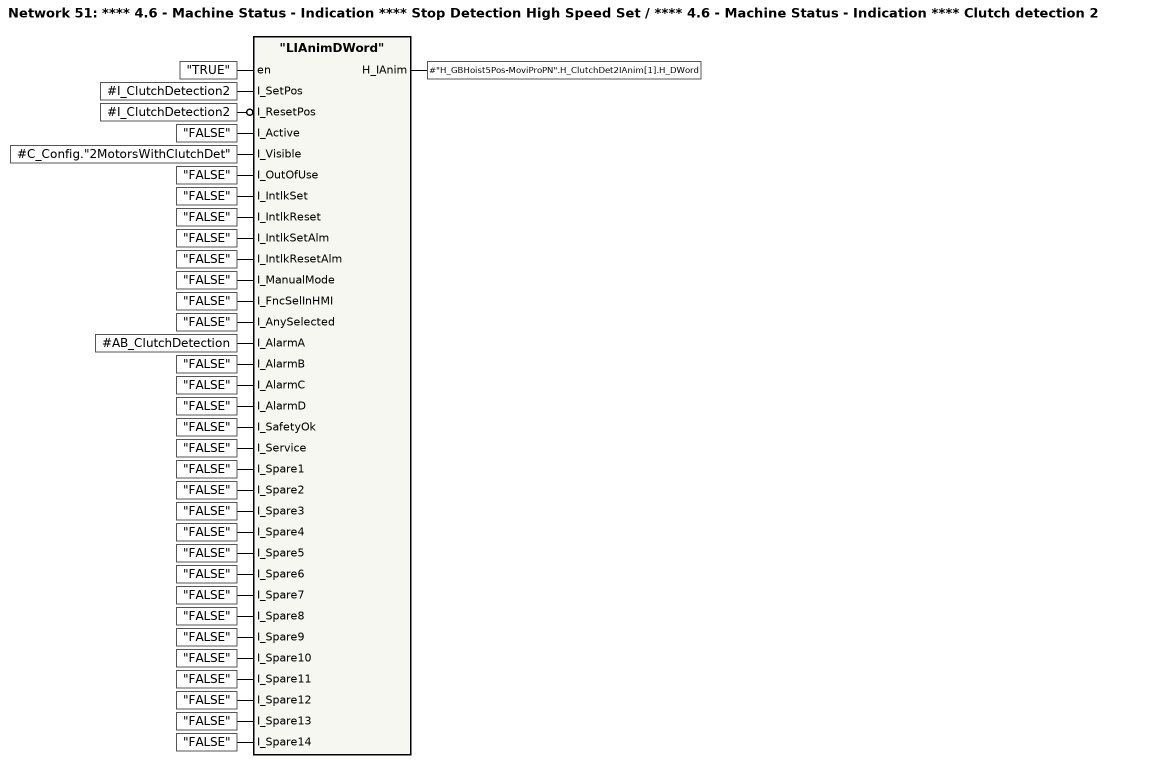
   IF "TRUE" THEN
       "LIAnimDWord"(I_SetPos := #I_ClutchDetection2,
                     I_ResetPos := NOT #I_ClutchDetection2,
                     I_Active := "FALSE",
                     I_Visible := #C_Config."2MotorsWithClutchDet",
                     I_OutOfUse := "FALSE",
                     I_IntlkSet := "FALSE",
                     I_IntlkReset := "FALSE",
                     I_IntlkSetAlm := "FALSE",
                     I_IntlkResetAlm := "FALSE",
                     I_ManualMode := "FALSE",
                     I_FncSelInHMI := "FALSE",
                     I_AnySelected := "FALSE",
                     I_AlarmA := #AB_ClutchDetection,
                     I_AlarmB := "FALSE",
                     I_AlarmC := "FALSE",
                     I_AlarmD := "FALSE",
                     I_SafetyOk := "FALSE",
                     I_Service := "FALSE",
                     I_Spare1 := "FALSE",
                     I_Spare2 := "FALSE",
                     I_Spare3 := "FALSE",
                     I_Spare4 := "FALSE",
                     I_Spare5 := "FALSE",
                     I_Spare6 := "FALSE",
                     I_Spare7 := "FALSE",
                     I_Spare8 := "FALSE",
                     I_Spare9 := "FALSE",
                     I_Spare10 := "FALSE",
                     I_Spare11 := "FALSE",
                     I_Spare12 := "FALSE",
                     I_Spare13 := "FALSE",
                     I_Spare14 := "FALSE",
                     H_IAnim => #"H_GBHoist5Pos-MoviProPN".H_ClutchDet2IAnim[1].H_DWord);
   END_IF;
END_REGION

REGION Network 52: **** 4.6 - Machine status - Indications **** Icon Animation
   // Animation for HMI
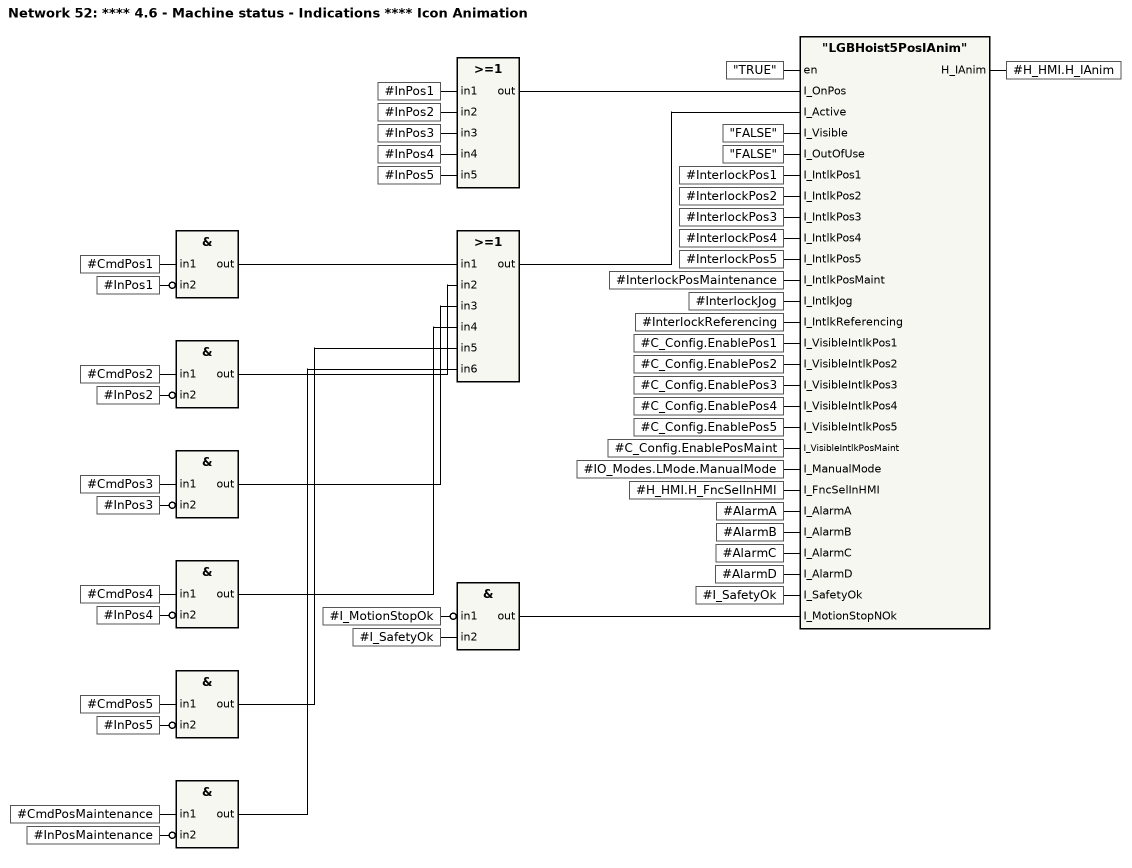
   IF "TRUE" THEN
       "LGBHoist5PosIAnim"(I_OnPos := #InPos1 OR #InPos2 OR #InPos3 OR #InPos4 OR #InPos5,
                           I_Active := (#CmdPos1 AND NOT #InPos1) OR (#CmdPos2 AND NOT #InPos2) OR (#CmdPos3 AND NOT #InPos3) OR (#CmdPos4 AND NOT #InPos4) OR (#CmdPos5 AND NOT #InPos5) OR (#CmdPosMaintenance AND NOT #InPosMaintenance),
                           I_Visible := "FALSE",
                           I_OutOfUse := "FALSE",
                           I_IntlkPos1 := #InterlockPos1,
                           I_IntlkPos2 := #InterlockPos2,
                           I_IntlkPos3 := #InterlockPos3,
                           I_IntlkPos4 := #InterlockPos4,
                           I_IntlkPos5 := #InterlockPos5,
                           I_IntlkPosMaint := #InterlockPosMaintenance,
                           I_IntlkJog := #InterlockJog,
                           I_IntlkReferencing := #InterlockReferencing,
                           I_VisibleIntlkPos1 := #C_Config.EnablePos1,
                           I_VisibleIntlkPos2 := #C_Config.EnablePos2,
                           I_VisibleIntlkPos3 := #C_Config.EnablePos3,
                           I_VisibleIntlkPos4 := #C_Config.EnablePos4,
                           I_VisibleIntlkPos5 := #C_Config.EnablePos5,
                           I_VisibleIntlkPosMaint := #C_Config.EnablePosMaint,
                           I_ManualMode := #IO_Modes.LMode.ManualMode,
                           I_FncSelInHMI := #H_HMI.H_FncSelInHMI,
                           I_AlarmA := #AlarmA,
                           I_AlarmB := #AlarmB,
                           I_AlarmC := #AlarmC,
                           I_AlarmD := #AlarmD,
                           I_SafetyOk := #I_SafetyOk,
                           I_MotionStopNOk := NOT #I_MotionStopOk AND #I_SafetyOk,
                           H_IAnim => #H_HMI.H_IAnim);
   END_IF;
END_REGION

REGION Network 53: **** 4.6 - Machine status - Indications **** Anim
   // Animation for HMI
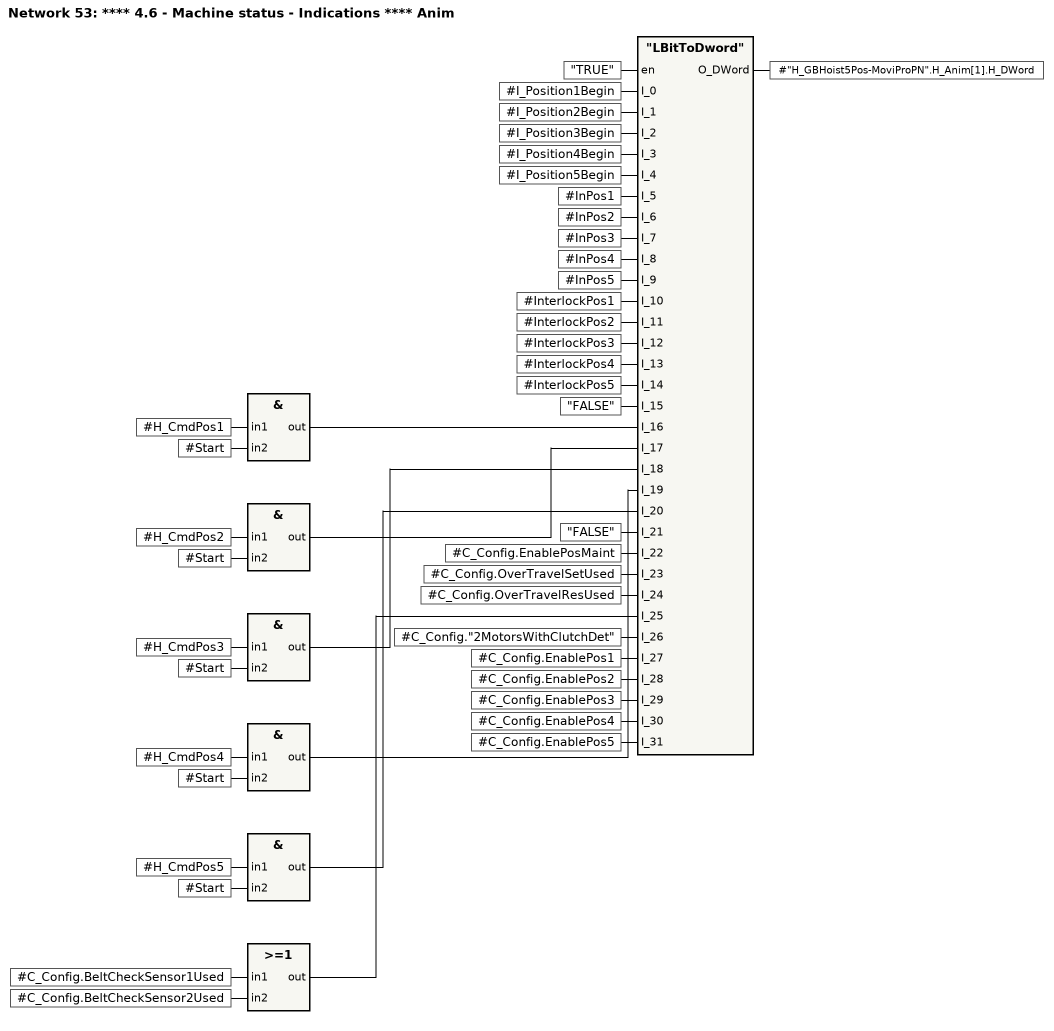
   IF "TRUE" THEN
       "LBitToDword"(I_0 := #I_Position1Begin,
                     I_1 := #I_Position2Begin,
                     I_2 := #I_Position3Begin,
                     I_3 := #I_Position4Begin,
                     I_4 := #I_Position5Begin,
                     I_5 := #InPos1,
                     I_6 := #InPos2,
                     I_7 := #InPos3,
                     I_8 := #InPos4,
                     I_9 := #InPos5,
                     I_10 := #InterlockPos1,
                     I_11 := #InterlockPos2,
                     I_12 := #InterlockPos3,
                     I_13 := #InterlockPos4,
                     I_14 := #InterlockPos5,
                     I_15 := "FALSE",
                     I_16 := #H_CmdPos1 AND #Start,
                     I_17 := #H_CmdPos2 AND #Start,
                     I_18 := #H_CmdPos3 AND #Start,
                     I_19 := #H_CmdPos4 AND #Start,
                     I_20 := #H_CmdPos5 AND #Start,
                     I_21 := "FALSE",
                     I_22 := #C_Config.EnablePosMaint,
                     I_23 := #C_Config.OverTravelSetUsed,
                     I_24 := #C_Config.OverTravelResUsed,
                     I_25 := #C_Config.BeltCheckSensor1Used OR #C_Config.BeltCheckSensor2Used,
                     I_26 := #C_Config."2MotorsWithClutchDet",
                     I_27 := #C_Config.EnablePos1,
                     I_28 := #C_Config.EnablePos2,
                     I_29 := #C_Config.EnablePos3,
                     I_30 := #C_Config.EnablePos4,
                     I_31 := #C_Config.EnablePos5,
                     O_DWord => #"H_GBHoist5Pos-MoviProPN".H_Anim[1].H_DWord);
   END_IF;
END_REGION

REGION Network 54: **** 4.6 - Machine status - Indications **** Anim
   // Animation for HMI
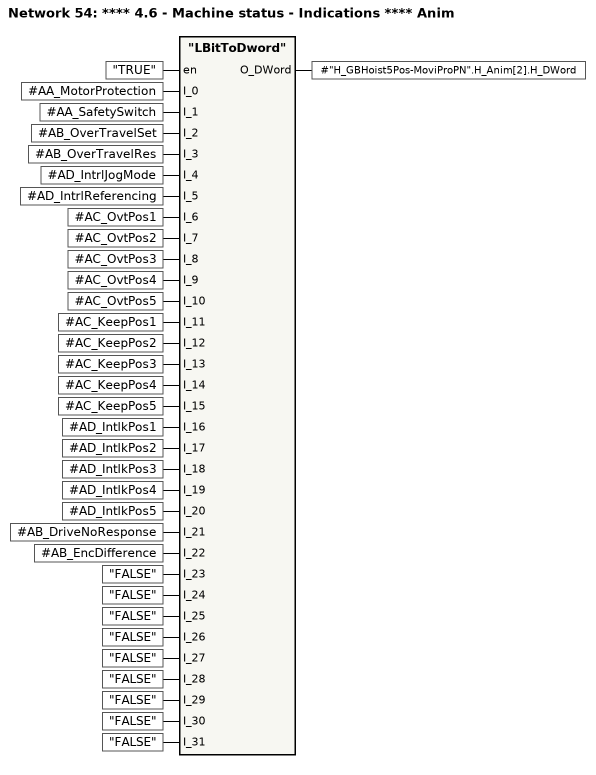
   IF "TRUE" THEN
       "LBitToDword"(I_0 := #AA_MotorProtection,
                     I_1 := #AA_SafetySwitch,
                     I_2 := #AB_OverTravelSet,
                     I_3 := #AB_OverTravelRes,
                     I_4 := #AD_IntrlJogMode,
                     I_5 := #AD_IntrlReferencing,
                     I_6 := #AC_OvtPos1,
                     I_7 := #AC_OvtPos2,
                     I_8 := #AC_OvtPos3,
                     I_9 := #AC_OvtPos4,
                     I_10 := #AC_OvtPos5,
                     I_11 := #AC_KeepPos1,
                     I_12 := #AC_KeepPos2,
                     I_13 := #AC_KeepPos3,
                     I_14 := #AC_KeepPos4,
                     I_15 := #AC_KeepPos5,
                     I_16 := #AD_IntlkPos1,
                     I_17 := #AD_IntlkPos2,
                     I_18 := #AD_IntlkPos3,
                     I_19 := #AD_IntlkPos4,
                     I_20 := #AD_IntlkPos5,
                     I_21 := #AB_DriveNoResponse,
                     I_22 := #AB_EncDifference,
                     I_23 := "FALSE",
                     I_24 := "FALSE",
                     I_25 := "FALSE",
                     I_26 := "FALSE",
                     I_27 := "FALSE",
                     I_28 := "FALSE",
                     I_29 := "FALSE",
                     I_30 := "FALSE",
                     I_31 := "FALSE",
                     O_DWord => #"H_GBHoist5Pos-MoviProPN".H_Anim[2].H_DWord);
   END_IF;
END_REGION

REGION Network 55: **** 4.6 - Machine status - Indications **** Anim
   // Animation for HMI
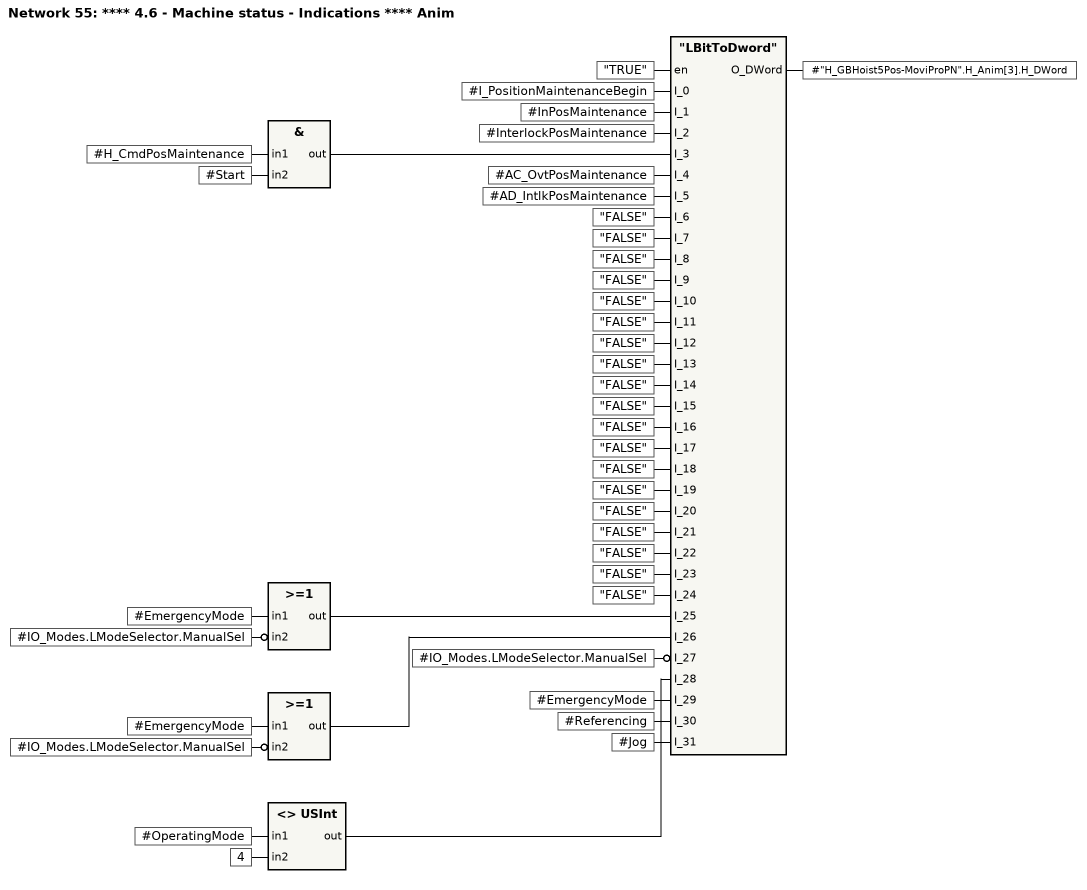
   IF "TRUE" THEN
       "LBitToDword"(I_0 := #I_PositionMaintenanceBegin,
                     I_1 := #InPosMaintenance,
                     I_2 := #InterlockPosMaintenance,
                     I_3 := #H_CmdPosMaintenance AND #Start,
                     I_4 := #AC_OvtPosMaintenance,
                     I_5 := #AD_IntlkPosMaintenance,
                     I_6 := "FALSE",
                     I_7 := "FALSE",
                     I_8 := "FALSE",
                     I_9 := "FALSE",
                     I_10 := "FALSE",
                     I_11 := "FALSE",
                     I_12 := "FALSE",
                     I_13 := "FALSE",
                     I_14 := "FALSE",
                     I_15 := "FALSE",
                     I_16 := "FALSE",
                     I_17 := "FALSE",
                     I_18 := "FALSE",
                     I_19 := "FALSE",
                     I_20 := "FALSE",
                     I_21 := "FALSE",
                     I_22 := "FALSE",
                     I_23 := "FALSE",
                     I_24 := "FALSE",
                     I_25 := #EmergencyMode OR NOT #IO_Modes.LModeSelector.ManualSel,
                     I_26 := #EmergencyMode OR NOT #IO_Modes.LModeSelector.ManualSel,
                     I_27 := NOT #IO_Modes.LModeSelector.ManualSel,
                     I_28 := #OperatingMode <> 4,
                     I_29 := #EmergencyMode,
                     I_30 := #Referencing,
                     I_31 := #Jog,
                     O_DWord => #"H_GBHoist5Pos-MoviProPN".H_Anim[3].H_DWord);
   END_IF;
END_REGION

REGION Network 56: **** 4.6 - Machine status - Indications **** Anim
   // Anim
